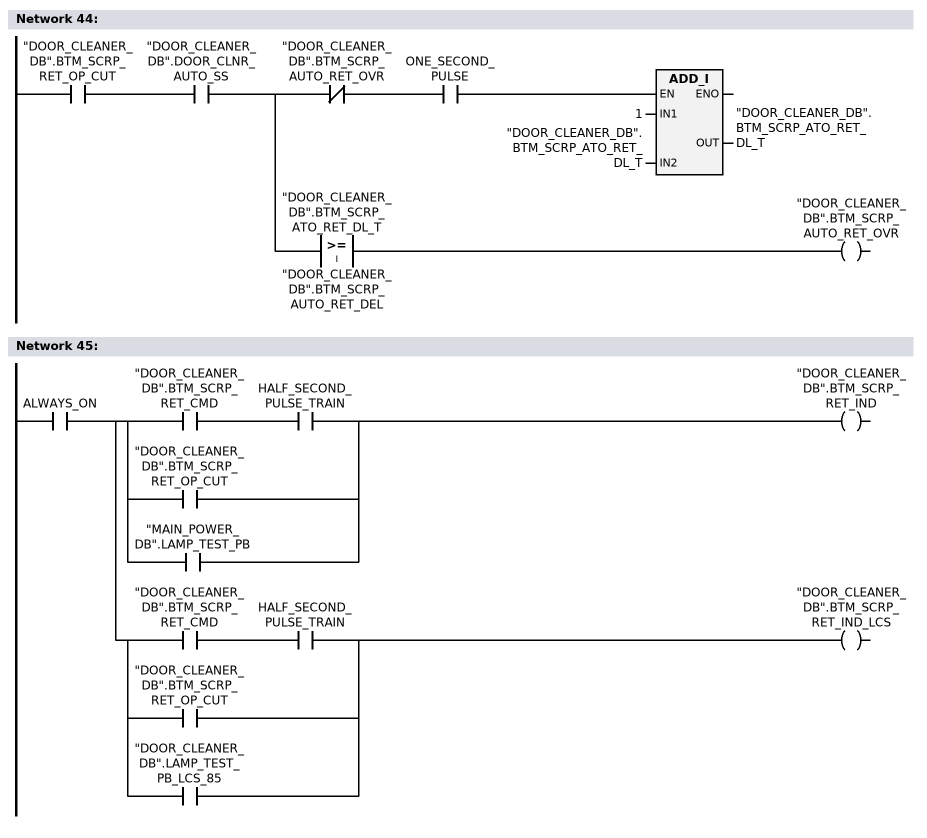
NETWORK
TITLE =
      A     "DOOR_CLEANER_DB".BTM_SCRP_RET_OP_CUT;
      A     "DOOR_CLEANER_DB".DOOR_CLNR_AUTO_SS;
      =     L 0.0;
      A     L 0.0;
      AN    "DOOR_CLEANER_DB".BTM_SCRP_AUTO_RET_OVR;
      A     "ONE_SECOND_PULSE";
      JNB   M042;
      L     1;
      L     "DOOR_CLEANER_DB".BTM_SCRP_ATO_RET_DL_T;
      +I;
      T     "DOOR_CLEANER_DB".BTM_SCRP_ATO_RET_DL_T;
M042: NOP   0;
      A     L 0.0;
      A(;
      L     "DOOR_CLEANER_DB".BTM_SCRP_ATO_RET_DL_T;
      L     "DOOR_CLEANER_DB".BTM_SCRP_AUTO_RET_DEL;
      >=I;
      );
      =     "DOOR_CLEANER_DB".BTM_SCRP_AUTO_RET_OVR;
NETWORK
TITLE =
      A     "ALWAYS_ON";
      =     L 0.0;
      A     L 0.0;
      A(;
      A     "DOOR_CLEANER_DB".BTM_SCRP_RET_CMD;
      A     "HALF_SECOND_PULSE_TRAIN";
      O     "DOOR_CLEANER_DB".BTM_SCRP_RET_OP_CUT;
      O     "MAIN_POWER_DB".LAMP_TEST_PB;
      );
      =     "DOOR_CLEANER_DB".BTM_SCRP_RET_IND;
      A     L 0.0;
      A(;
      A     "DOOR_CLEANER_DB".BTM_SCRP_RET_CMD;
      A     "HALF_SECOND_PULSE_TRAIN";
      O     "DOOR_CLEANER_DB".BTM_SCRP_RET_OP_CUT;
      O     "DOOR_CLEANER_DB".LAMP_TEST_PB_LCS_85;
      );
      =     "DOOR_CLEANER_DB".BTM_SCRP_RET_IND_LCS;
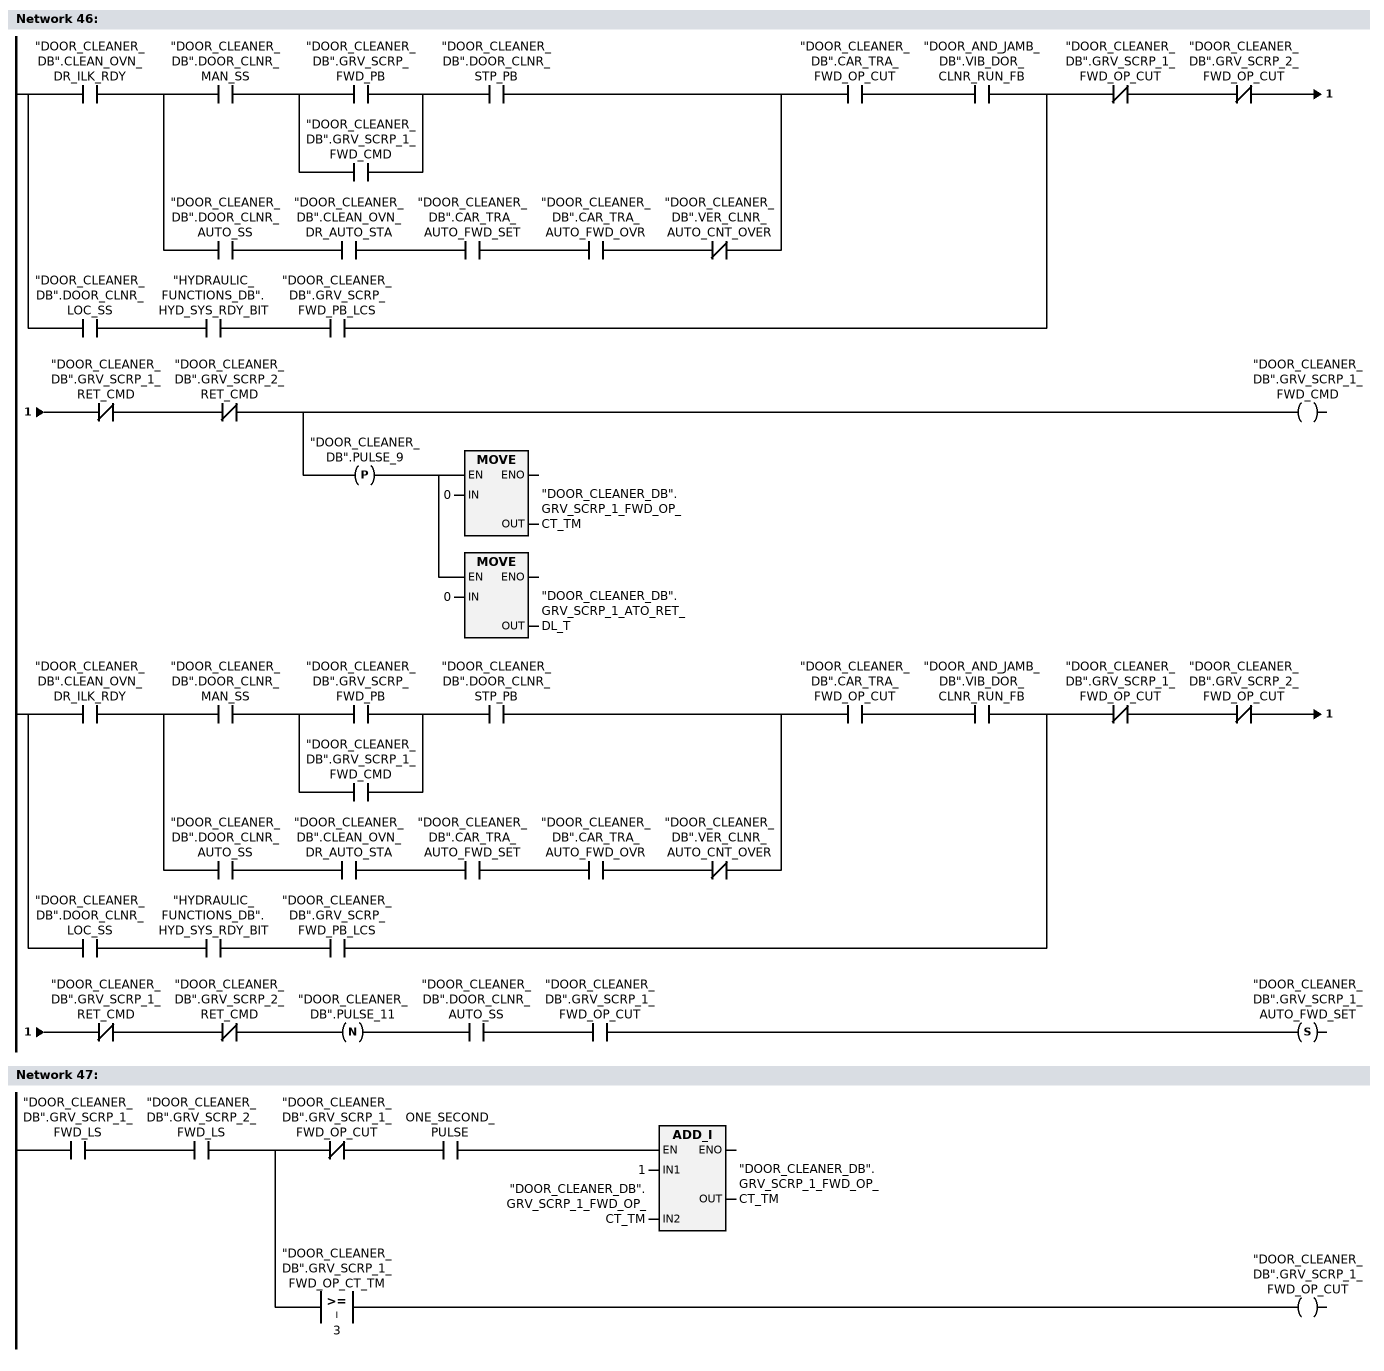
NETWORK
TITLE =
      A(;
      A     "DOOR_CLEANER_DB".CLEAN_OVN_DR_ILK_RDY;
      A(;
      A     "DOOR_CLEANER_DB".DOOR_CLNR_MAN_SS;
      A(;
      O     "DOOR_CLEANER_DB".GRV_SCRP_FWD_PB;
      O     "DOOR_CLEANER_DB".GRV_SCRP_1_FWD_CMD;
      );
      A     "DOOR_CLEANER_DB".DOOR_CLNR_STP_PB;
      O;
      A     "DOOR_CLEANER_DB".DOOR_CLNR_AUTO_SS;
      A     "DOOR_CLEANER_DB".CLEAN_OVN_DR_AUTO_STA;
      A     "DOOR_CLEANER_DB".CAR_TRA_AUTO_FWD_SET;
      A     "DOOR_CLEANER_DB".CAR_TRA_AUTO_FWD_OVR;
      AN    "DOOR_CLEANER_DB".VER_CLNR_AUTO_CNT_OVER;
      );
      A     "DOOR_CLEANER_DB".CAR_TRA_FWD_OP_CUT;
      A     "DOOR_AND_JAMB_DB".VIB_DOR_CLNR_RUN_FB;
      O;
      A     "DOOR_CLEANER_DB".DOOR_CLNR_LOC_SS;
      A     "HYDRAULIC_FUNCTIONS_DB".HYD_SYS_RDY_BIT;
      A     "DOOR_CLEANER_DB".GRV_SCRP_FWD_PB_LCS;
      );
      AN    "DOOR_CLEANER_DB".GRV_SCRP_1_FWD_OP_CUT;
      AN    "DOOR_CLEANER_DB".GRV_SCRP_2_FWD_OP_CUT;
      AN    "DOOR_CLEANER_DB".GRV_SCRP_1_RET_CMD;
      AN    "DOOR_CLEANER_DB".GRV_SCRP_2_RET_CMD;
      =     L 0.0;
      A     L 0.0;
      BLD   102;
      =     "DOOR_CLEANER_DB".GRV_SCRP_1_FWD_CMD;
      A(;
      A     L 0.0;
      FN    "DOOR_CLEANER_DB".PULSE_11;
      );
      A     "DOOR_CLEANER_DB".DOOR_CLNR_AUTO_SS;
      A     "DOOR_CLEANER_DB".GRV_SCRP_1_FWD_OP_CUT;
      S     "DOOR_CLEANER_DB".GRV_SCRP_1_AUTO_FWD_SET;
      A     L 0.0;
      FP    "DOOR_CLEANER_DB".PULSE_9;
      =     L 0.1;
      A     L 0.1;
      JNB   M043;
      L     0;
      T     "DOOR_CLEANER_DB".GRV_SCRP_1_FWD_OP_CT_TM;
M043: NOP   0;
      A     L 0.1;
      JNB   M044;
      L     0;
      T     "DOOR_CLEANER_DB".GRV_SCRP_1_ATO_RET_DL_T;
M044: NOP   0;
NETWORK
TITLE =
      A     "DOOR_CLEANER_DB".GRV_SCRP_1_FWD_LS;
      A     "DOOR_CLEANER_DB".GRV_SCRP_2_FWD_LS;
      =     L 0.0;
      A     L 0.0;
      AN    "DOOR_CLEANER_DB".GRV_SCRP_1_FWD_OP_CUT;
      A     "ONE_SECOND_PULSE";
      JNB   M045;
      L     1;
      L     "DOOR_CLEANER_DB".GRV_SCRP_1_FWD_OP_CT_TM;
      +I;
      T     "DOOR_CLEANER_DB".GRV_SCRP_1_FWD_OP_CT_TM;
M045: NOP   0;
      A     L 0.0;
      A(;
      L     "DOOR_CLEANER_DB".GRV_SCRP_1_FWD_OP_CT_TM;
      L     3;
      >=I;
      );
      =     "DOOR_CLEANER_DB".GRV_SCRP_1_FWD_OP_CUT;
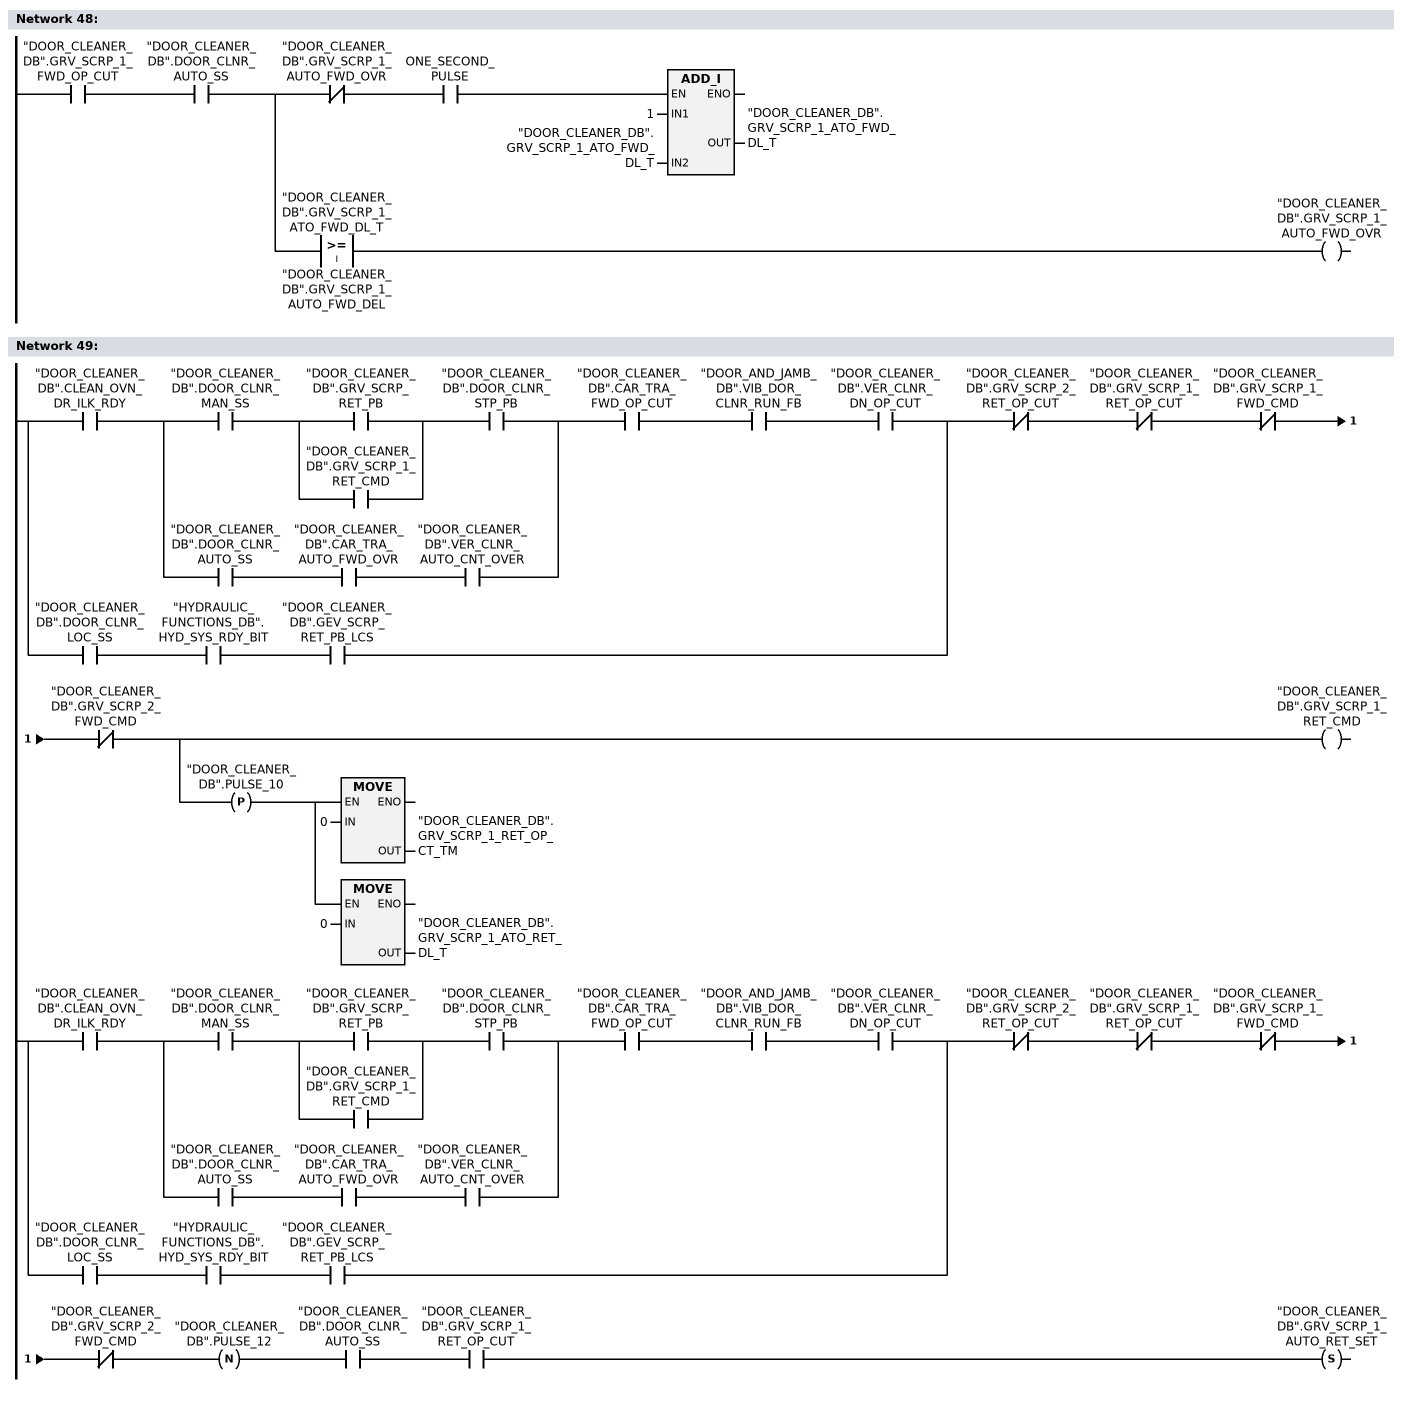
NETWORK
TITLE =
      A     "DOOR_CLEANER_DB".GRV_SCRP_1_FWD_OP_CUT;
      A     "DOOR_CLEANER_DB".DOOR_CLNR_AUTO_SS;
      =     L 0.0;
      A     L 0.0;
      AN    "DOOR_CLEANER_DB".GRV_SCRP_1_AUTO_FWD_OVR;
      A     "ONE_SECOND_PULSE";
      JNB   M046;
      L     1;
      L     "DOOR_CLEANER_DB".GRV_SCRP_1_ATO_FWD_DL_T;
      +I;
      T     "DOOR_CLEANER_DB".GRV_SCRP_1_ATO_FWD_DL_T;
M046: NOP   0;
      A     L 0.0;
      A(;
      L     "DOOR_CLEANER_DB".GRV_SCRP_1_ATO_FWD_DL_T;
      L     "DOOR_CLEANER_DB".GRV_SCRP_1_AUTO_FWD_DEL;
      >=I;
      );
      =     "DOOR_CLEANER_DB".GRV_SCRP_1_AUTO_FWD_OVR;
NETWORK
TITLE =
      A(;
      A     "DOOR_CLEANER_DB".CLEAN_OVN_DR_ILK_RDY;
      A(;
      A     "DOOR_CLEANER_DB".DOOR_CLNR_MAN_SS;
      A(;
      O     "DOOR_CLEANER_DB".GRV_SCRP_RET_PB;
      O     "DOOR_CLEANER_DB".GRV_SCRP_1_RET_CMD;
      );
      A     "DOOR_CLEANER_DB".DOOR_CLNR_STP_PB;
      O;
      A     "DOOR_CLEANER_DB".DOOR_CLNR_AUTO_SS;
      A     "DOOR_CLEANER_DB".CAR_TRA_AUTO_FWD_OVR;
      A     "DOOR_CLEANER_DB".VER_CLNR_AUTO_CNT_OVER;
      );
      A     "DOOR_CLEANER_DB".CAR_TRA_FWD_OP_CUT;
      A     "DOOR_AND_JAMB_DB".VIB_DOR_CLNR_RUN_FB;
      A     "DOOR_CLEANER_DB".VER_CLNR_DN_OP_CUT;
      O;
      A     "DOOR_CLEANER_DB".DOOR_CLNR_LOC_SS;
      A     "HYDRAULIC_FUNCTIONS_DB".HYD_SYS_RDY_BIT;
      A     "DOOR_CLEANER_DB".GEV_SCRP_RET_PB_LCS;
      );
      AN    "DOOR_CLEANER_DB".GRV_SCRP_2_RET_OP_CUT;
      AN    "DOOR_CLEANER_DB".GRV_SCRP_1_RET_OP_CUT;
      AN    "DOOR_CLEANER_DB".GRV_SCRP_1_FWD_CMD;
      AN    "DOOR_CLEANER_DB".GRV_SCRP_2_FWD_CMD;
      =     L 0.0;
      A     L 0.0;
      BLD   102;
      =     "DOOR_CLEANER_DB".GRV_SCRP_1_RET_CMD;
      A(;
      A     L 0.0;
      FN    "DOOR_CLEANER_DB".PULSE_12;
      );
      A     "DOOR_CLEANER_DB".DOOR_CLNR_AUTO_SS;
      A     "DOOR_CLEANER_DB".GRV_SCRP_1_RET_OP_CUT;
      S     "DOOR_CLEANER_DB".GRV_SCRP_1_AUTO_RET_SET;
      A     L 0.0;
      FP    "DOOR_CLEANER_DB".PULSE_10;
      =     L 0.1;
      A     L 0.1;
      JNB   M047;
      L     0;
      T     "DOOR_CLEANER_DB".GRV_SCRP_1_RET_OP_CT_TM;
M047: NOP   0;
      A     L 0.1;
      JNB   M048;
      L     0;
      T     "DOOR_CLEANER_DB".GRV_SCRP_1_ATO_RET_DL_T;
M048: NOP   0;
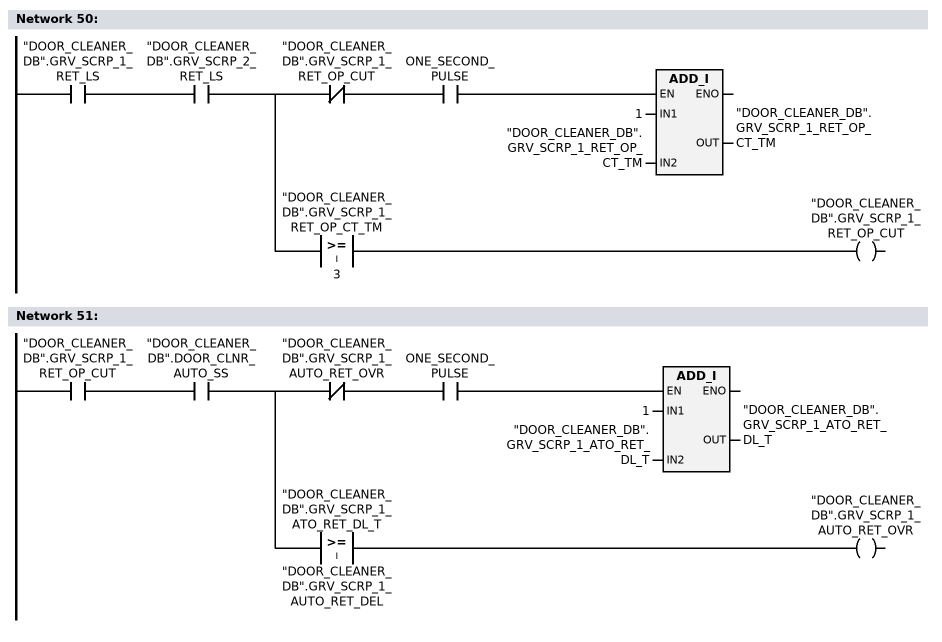
NETWORK
TITLE =
      A     "DOOR_CLEANER_DB".GRV_SCRP_1_RET_LS;
      A     "DOOR_CLEANER_DB".GRV_SCRP_2_RET_LS;
      =     L 0.0;
      A     L 0.0;
      AN    "DOOR_CLEANER_DB".GRV_SCRP_1_RET_OP_CUT;
      A     "ONE_SECOND_PULSE";
      JNB   M049;
      L     1;
      L     "DOOR_CLEANER_DB".GRV_SCRP_1_RET_OP_CT_TM;
      +I;
      T     "DOOR_CLEANER_DB".GRV_SCRP_1_RET_OP_CT_TM;
M049: NOP   0;
      A     L 0.0;
      A(;
      L     "DOOR_CLEANER_DB".GRV_SCRP_1_RET_OP_CT_TM;
      L     3;
      >=I;
      );
      =     "DOOR_CLEANER_DB".GRV_SCRP_1_RET_OP_CUT;
NETWORK
TITLE =
      A     "DOOR_CLEANER_DB".GRV_SCRP_1_RET_OP_CUT;
      A     "DOOR_CLEANER_DB".DOOR_CLNR_AUTO_SS;
      =     L 0.0;
      A     L 0.0;
      AN    "DOOR_CLEANER_DB".GRV_SCRP_1_AUTO_RET_OVR;
      A     "ONE_SECOND_PULSE";
      JNB   M050;
      L     1;
      L     "DOOR_CLEANER_DB".GRV_SCRP_1_ATO_RET_DL_T;
      +I;
      T     "DOOR_CLEANER_DB".GRV_SCRP_1_ATO_RET_DL_T;
M050: NOP   0;
      A     L 0.0;
      A(;
      L     "DOOR_CLEANER_DB".GRV_SCRP_1_ATO_RET_DL_T;
      L     "DOOR_CLEANER_DB".GRV_SCRP_1_AUTO_RET_DEL;
      >=I;
      );
      =     "DOOR_CLEANER_DB".GRV_SCRP_1_AUTO_RET_OVR;
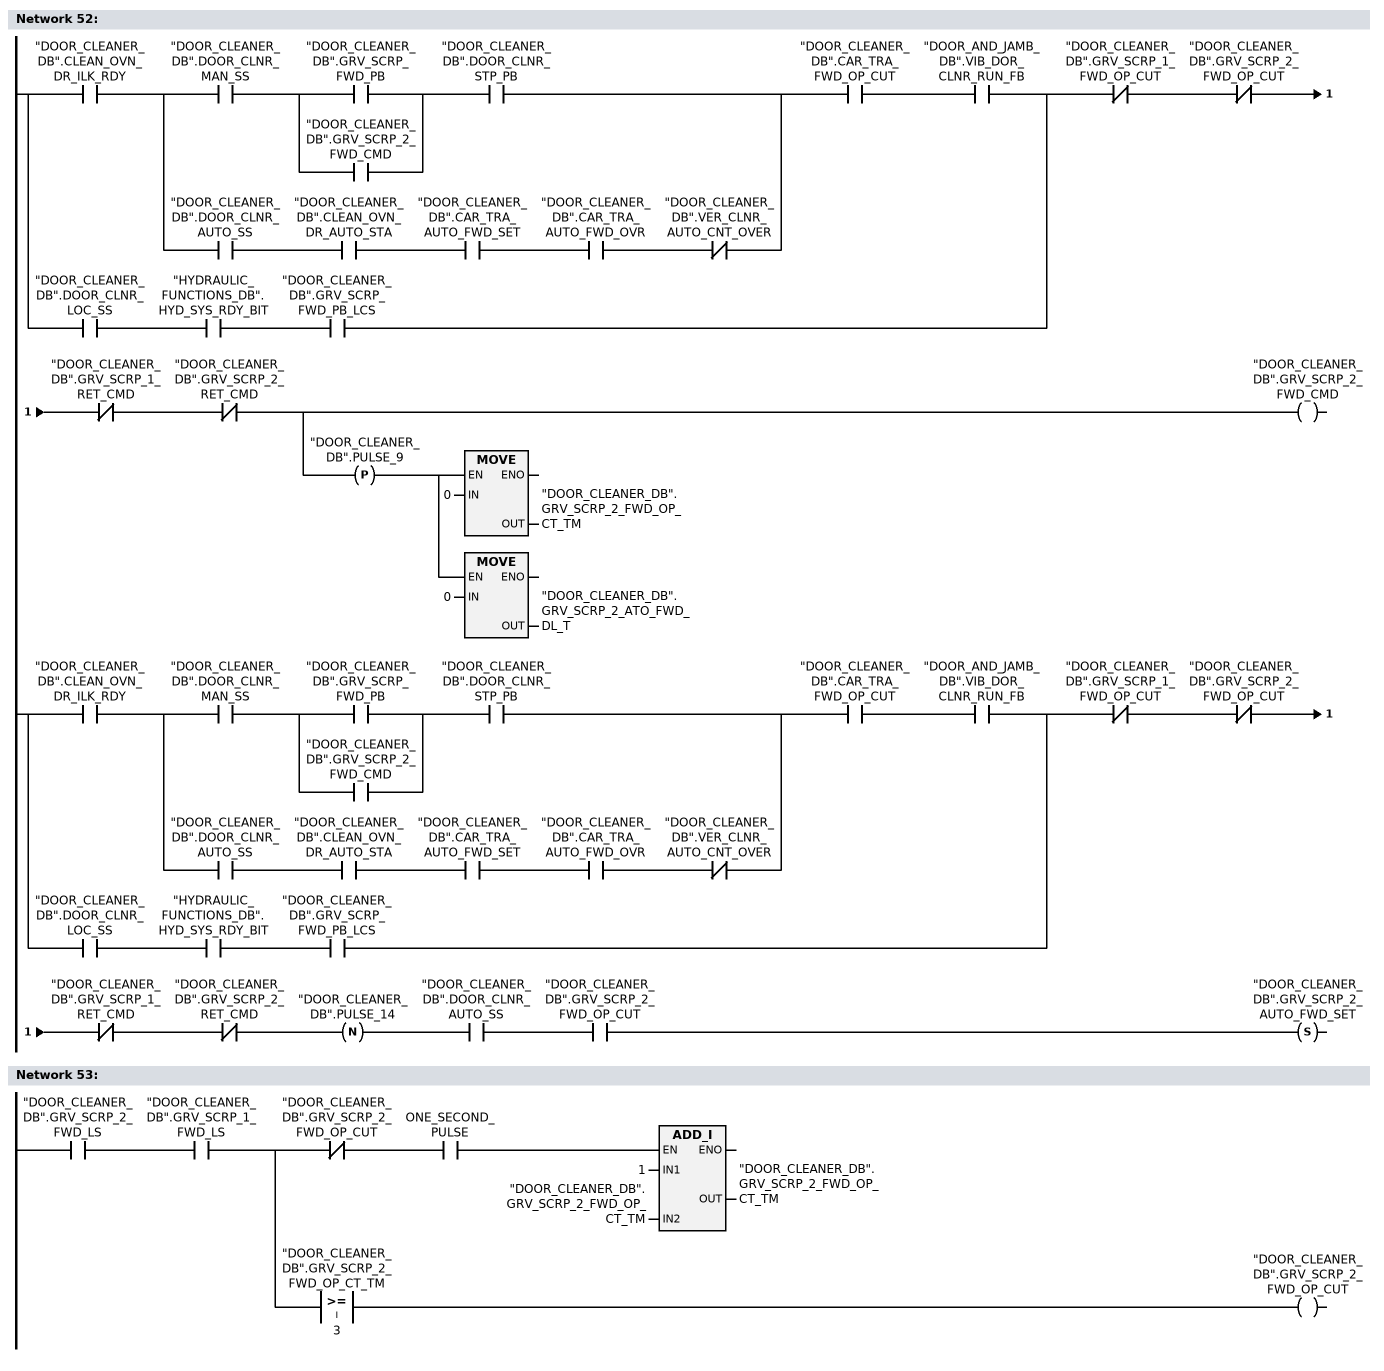
NETWORK
TITLE =
      A(;
      A     "DOOR_CLEANER_DB".CLEAN_OVN_DR_ILK_RDY;
      A(;
      A     "DOOR_CLEANER_DB".DOOR_CLNR_MAN_SS;
      A(;
      O     "DOOR_CLEANER_DB".GRV_SCRP_FWD_PB;
      O     "DOOR_CLEANER_DB".GRV_SCRP_2_FWD_CMD;
      );
      A     "DOOR_CLEANER_DB".DOOR_CLNR_STP_PB;
      O;
      A     "DOOR_CLEANER_DB".DOOR_CLNR_AUTO_SS;
      A     "DOOR_CLEANER_DB".CLEAN_OVN_DR_AUTO_STA;
      A     "DOOR_CLEANER_DB".CAR_TRA_AUTO_FWD_SET;
      A     "DOOR_CLEANER_DB".CAR_TRA_AUTO_FWD_OVR;
      AN    "DOOR_CLEANER_DB".VER_CLNR_AUTO_CNT_OVER;
      );
      A     "DOOR_CLEANER_DB".CAR_TRA_FWD_OP_CUT;
      A     "DOOR_AND_JAMB_DB".VIB_DOR_CLNR_RUN_FB;
      O;
      A     "DOOR_CLEANER_DB".DOOR_CLNR_LOC_SS;
      A     "HYDRAULIC_FUNCTIONS_DB".HYD_SYS_RDY_BIT;
      A     "DOOR_CLEANER_DB".GRV_SCRP_FWD_PB_LCS;
      );
      AN    "DOOR_CLEANER_DB".GRV_SCRP_1_FWD_OP_CUT;
      AN    "DOOR_CLEANER_DB".GRV_SCRP_2_FWD_OP_CUT;
      AN    "DOOR_CLEANER_DB".GRV_SCRP_1_RET_CMD;
      AN    "DOOR_CLEANER_DB".GRV_SCRP_2_RET_CMD;
      =     L 0.0;
      A     L 0.0;
      BLD   102;
      =     "DOOR_CLEANER_DB".GRV_SCRP_2_FWD_CMD;
      A(;
      A     L 0.0;
      FN    "DOOR_CLEANER_DB".PULSE_14;
      );
      A     "DOOR_CLEANER_DB".DOOR_CLNR_AUTO_SS;
      A     "DOOR_CLEANER_DB".GRV_SCRP_2_FWD_OP_CUT;
      S     "DOOR_CLEANER_DB".GRV_SCRP_2_AUTO_FWD_SET;
      A     L 0.0;
      FP    "DOOR_CLEANER_DB".PULSE_9;
      =     L 0.1;
      A     L 0.1;
      JNB   M051;
      L     0;
      T     "DOOR_CLEANER_DB".GRV_SCRP_2_FWD_OP_CT_TM;
M051: NOP   0;
      A     L 0.1;
      JNB   M052;
      L     0;
      T     "DOOR_CLEANER_DB".GRV_SCRP_2_ATO_FWD_DL_T;
M052: NOP   0;
NETWORK
TITLE =
      A     "DOOR_CLEANER_DB".GRV_SCRP_2_FWD_LS;
      A     "DOOR_CLEANER_DB".GRV_SCRP_1_FWD_LS;
      =     L 0.0;
      A     L 0.0;
      AN    "DOOR_CLEANER_DB".GRV_SCRP_2_FWD_OP_CUT;
      A     "ONE_SECOND_PULSE";
      JNB   M053;
      L     1;
      L     "DOOR_CLEANER_DB".GRV_SCRP_2_FWD_OP_CT_TM;
      +I;
      T     "DOOR_CLEANER_DB".GRV_SCRP_2_FWD_OP_CT_TM;
M053: NOP   0;
      A     L 0.0;
      A(;
      L     "DOOR_CLEANER_DB".GRV_SCRP_2_FWD_OP_CT_TM;
      L     3;
      >=I;
      );
      =     "DOOR_CLEANER_DB".GRV_SCRP_2_FWD_OP_CUT;
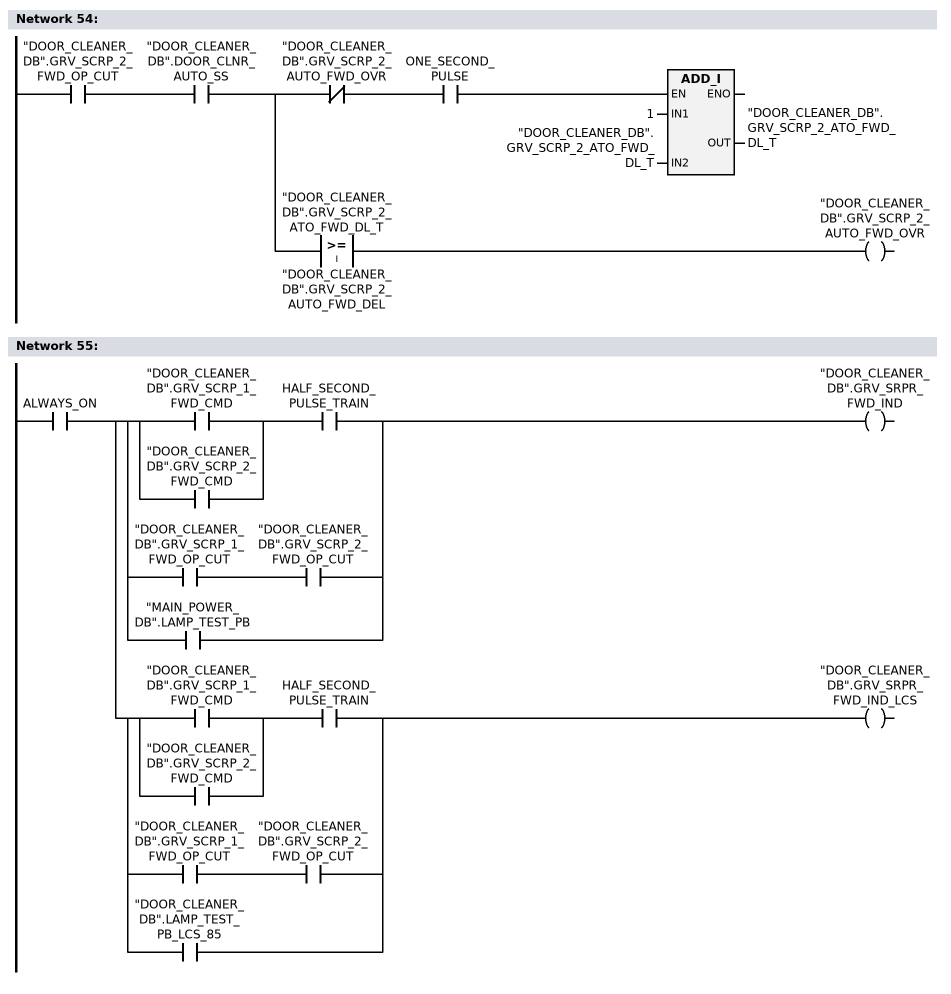
NETWORK
TITLE =
      A     "DOOR_CLEANER_DB".GRV_SCRP_2_FWD_OP_CUT;
      A     "DOOR_CLEANER_DB".DOOR_CLNR_AUTO_SS;
      =     L 0.0;
      A     L 0.0;
      AN    "DOOR_CLEANER_DB".GRV_SCRP_2_AUTO_FWD_OVR;
      A     "ONE_SECOND_PULSE";
      JNB   M054;
      L     1;
      L     "DOOR_CLEANER_DB".GRV_SCRP_2_ATO_FWD_DL_T;
      +I;
      T     "DOOR_CLEANER_DB".GRV_SCRP_2_ATO_FWD_DL_T;
M054: NOP   0;
      A     L 0.0;
      A(;
      L     "DOOR_CLEANER_DB".GRV_SCRP_2_ATO_FWD_DL_T;
      L     "DOOR_CLEANER_DB".GRV_SCRP_2_AUTO_FWD_DEL;
      >=I;
      );
      =     "DOOR_CLEANER_DB".GRV_SCRP_2_AUTO_FWD_OVR;
NETWORK
TITLE =
      A     "ALWAYS_ON";
      =     L 0.0;
      A     L 0.0;
      A(;
      A(;
      O     "DOOR_CLEANER_DB".GRV_SCRP_1_FWD_CMD;
      O     "DOOR_CLEANER_DB".GRV_SCRP_2_FWD_CMD;
      );
      A     "HALF_SECOND_PULSE_TRAIN";
      O;
      A     "DOOR_CLEANER_DB".GRV_SCRP_1_FWD_OP_CUT;
      A     "DOOR_CLEANER_DB".GRV_SCRP_2_FWD_OP_CUT;
      O     "MAIN_POWER_DB".LAMP_TEST_PB;
      );
      =     "DOOR_CLEANER_DB".GRV_SRPR_FWD_IND;
      A     L 0.0;
      A(;
      A(;
      O     "DOOR_CLEANER_DB".GRV_SCRP_1_FWD_CMD;
      O     "DOOR_CLEANER_DB".GRV_SCRP_2_FWD_CMD;
      );
      A     "HALF_SECOND_PULSE_TRAIN";
      O;
      A     "DOOR_CLEANER_DB".GRV_SCRP_1_FWD_OP_CUT;
      A     "DOOR_CLEANER_DB".GRV_SCRP_2_FWD_OP_CUT;
      O     "DOOR_CLEANER_DB".LAMP_TEST_PB_LCS_85;
      );
      =     "DOOR_CLEANER_DB".GRV_SRPR_FWD_IND_LCS;
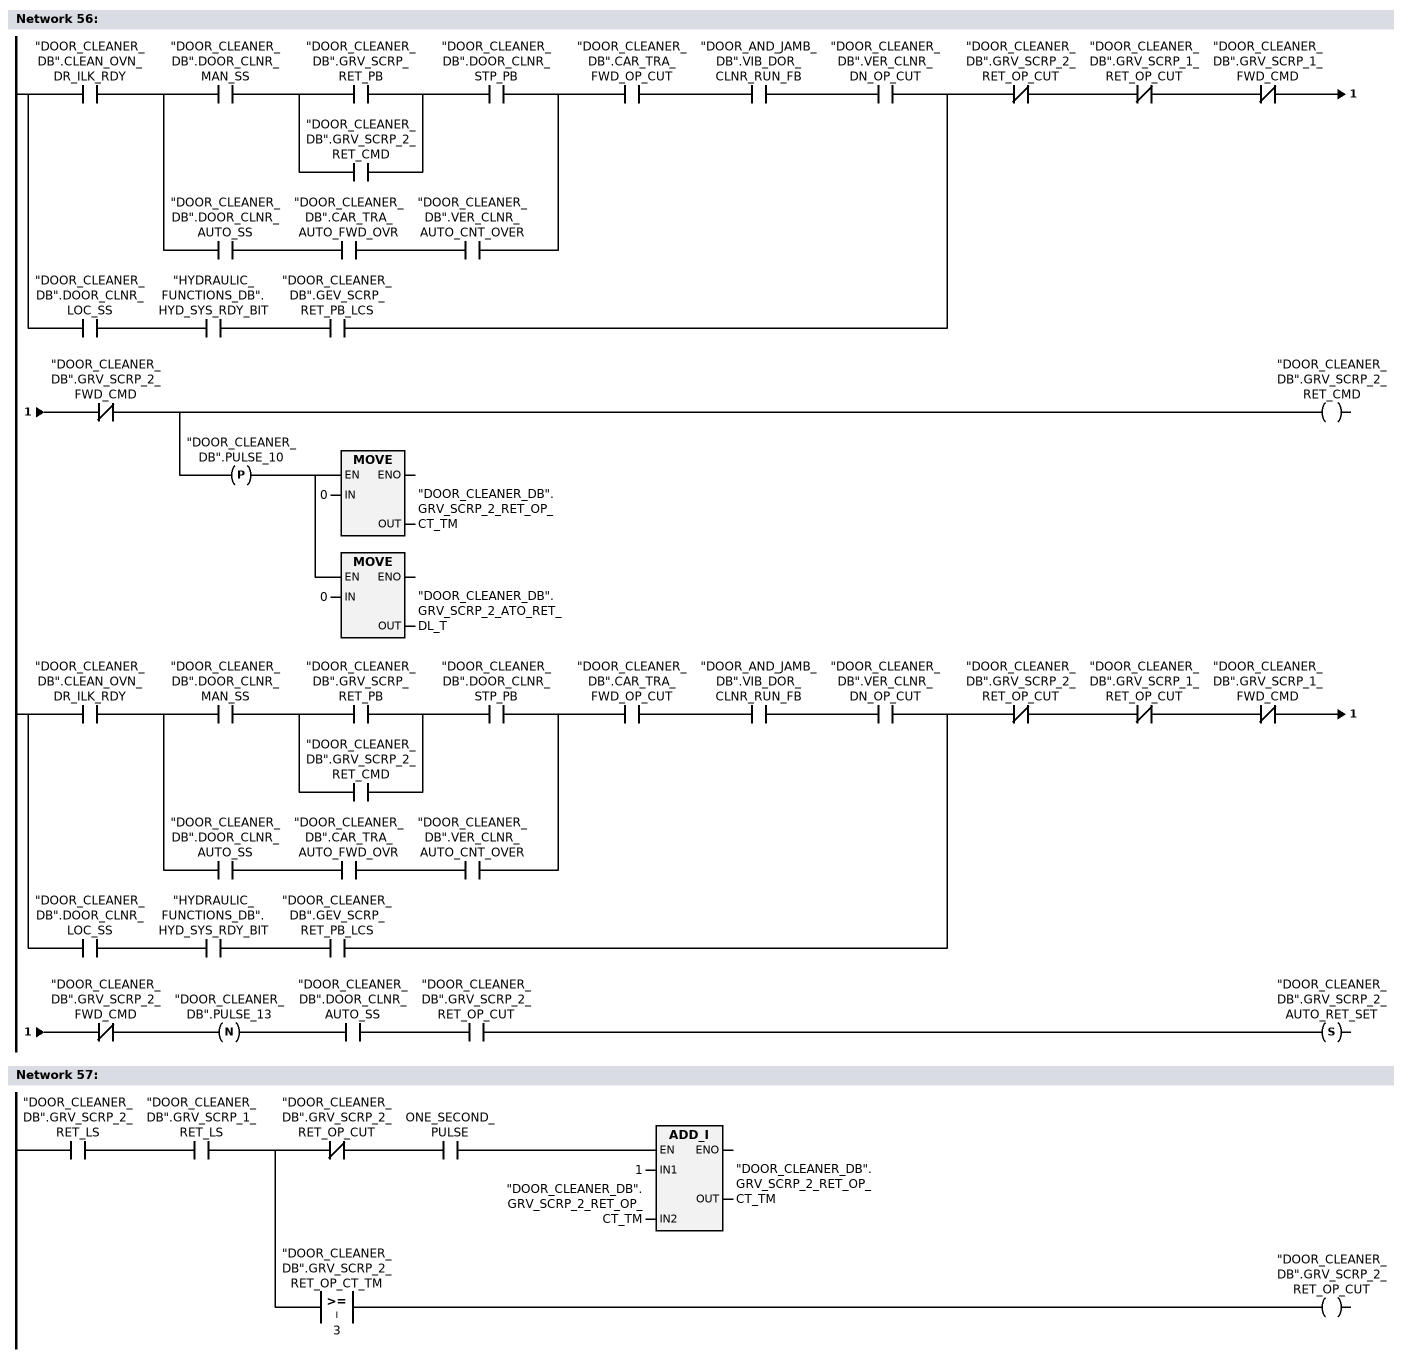
NETWORK
TITLE =
      A(;
      A     "DOOR_CLEANER_DB".CLEAN_OVN_DR_ILK_RDY;
      A(;
      A     "DOOR_CLEANER_DB".DOOR_CLNR_MAN_SS;
      A(;
      O     "DOOR_CLEANER_DB".GRV_SCRP_RET_PB;
      O     "DOOR_CLEANER_DB".GRV_SCRP_2_RET_CMD;
      );
      A     "DOOR_CLEANER_DB".DOOR_CLNR_STP_PB;
      O;
      A     "DOOR_CLEANER_DB".DOOR_CLNR_AUTO_SS;
      A     "DOOR_CLEANER_DB".CAR_TRA_AUTO_FWD_OVR;
      A     "DOOR_CLEANER_DB".VER_CLNR_AUTO_CNT_OVER;
      );
      A     "DOOR_CLEANER_DB".CAR_TRA_FWD_OP_CUT;
      A     "DOOR_AND_JAMB_DB".VIB_DOR_CLNR_RUN_FB;
      A     "DOOR_CLEANER_DB".VER_CLNR_DN_OP_CUT;
      O;
      A     "DOOR_CLEANER_DB".DOOR_CLNR_LOC_SS;
      A     "HYDRAULIC_FUNCTIONS_DB".HYD_SYS_RDY_BIT;
      A     "DOOR_CLEANER_DB".GEV_SCRP_RET_PB_LCS;
      );
      AN    "DOOR_CLEANER_DB".GRV_SCRP_2_RET_OP_CUT;
      AN    "DOOR_CLEANER_DB".GRV_SCRP_1_RET_OP_CUT;
      AN    "DOOR_CLEANER_DB".GRV_SCRP_1_FWD_CMD;
      AN    "DOOR_CLEANER_DB".GRV_SCRP_2_FWD_CMD;
      =     L 0.0;
      A     L 0.0;
      BLD   102;
      =     "DOOR_CLEANER_DB".GRV_SCRP_2_RET_CMD;
      A(;
      A     L 0.0;
      FN    "DOOR_CLEANER_DB".PULSE_13;
      );
      A     "DOOR_CLEANER_DB".DOOR_CLNR_AUTO_SS;
      A     "DOOR_CLEANER_DB".GRV_SCRP_2_RET_OP_CUT;
      S     "DOOR_CLEANER_DB".GRV_SCRP_2_AUTO_RET_SET;
      A     L 0.0;
      FP    "DOOR_CLEANER_DB".PULSE_10;
      =     L 0.1;
      A     L 0.1;
      JNB   M055;
      L     0;
      T     "DOOR_CLEANER_DB".GRV_SCRP_2_RET_OP_CT_TM;
M055: NOP   0;
      A     L 0.1;
      JNB   M056;
      L     0;
      T     "DOOR_CLEANER_DB".GRV_SCRP_2_ATO_RET_DL_T;
M056: NOP   0;
NETWORK
TITLE =
      A     "DOOR_CLEANER_DB".GRV_SCRP_2_RET_LS;
      A     "DOOR_CLEANER_DB".GRV_SCRP_1_RET_LS;
      =     L 0.0;
      A     L 0.0;
      AN    "DOOR_CLEANER_DB".GRV_SCRP_2_RET_OP_CUT;
      A     "ONE_SECOND_PULSE";
      JNB   M057;
      L     1;
      L     "DOOR_CLEANER_DB".GRV_SCRP_2_RET_OP_CT_TM;
      +I;
      T     "DOOR_CLEANER_DB".GRV_SCRP_2_RET_OP_CT_TM;
M057: NOP   0;
      A     L 0.0;
      A(;
      L     "DOOR_CLEANER_DB".GRV_SCRP_2_RET_OP_CT_TM;
      L     3;
      >=I;
      );
      =     "DOOR_CLEANER_DB".GRV_SCRP_2_RET_OP_CUT;
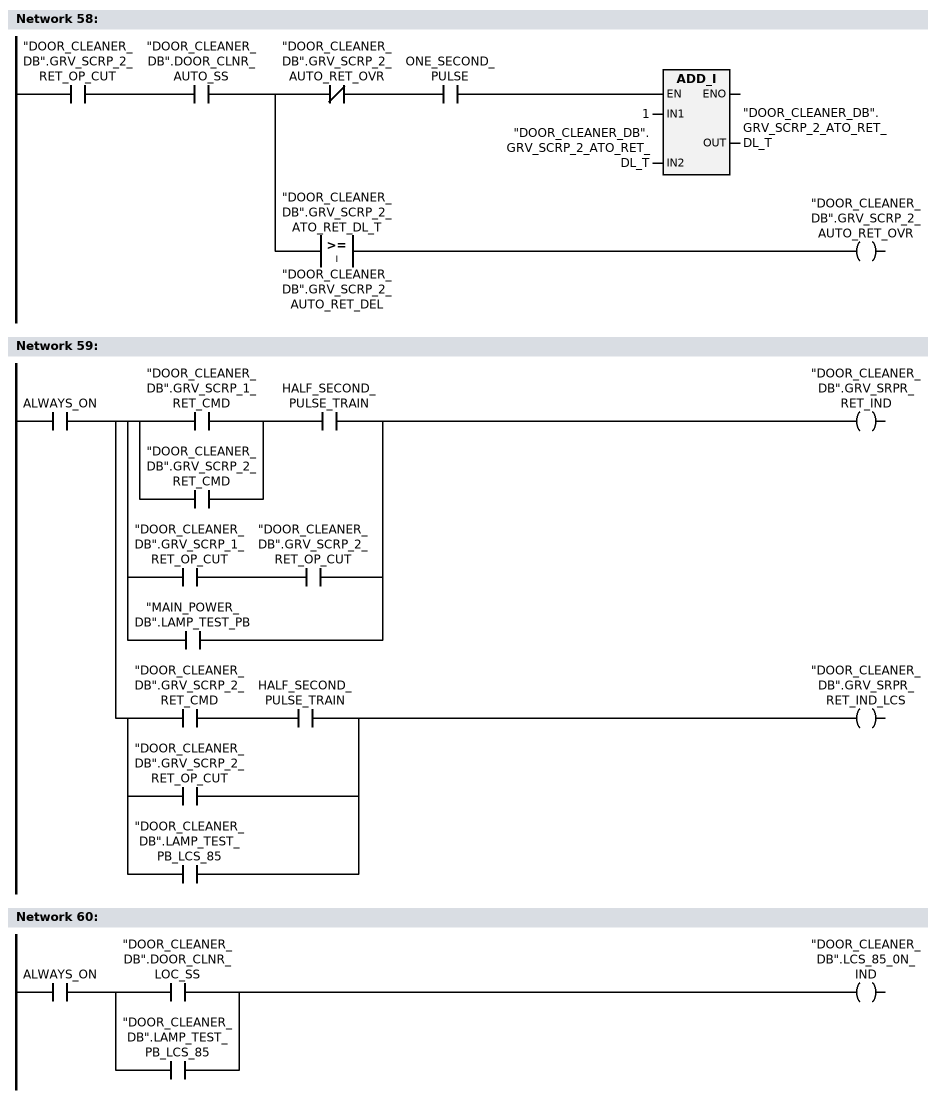
NETWORK
TITLE =
      A     "DOOR_CLEANER_DB".GRV_SCRP_2_RET_OP_CUT;
      A     "DOOR_CLEANER_DB".DOOR_CLNR_AUTO_SS;
      =     L 0.0;
      A     L 0.0;
      AN    "DOOR_CLEANER_DB".GRV_SCRP_2_AUTO_RET_OVR;
      A     "ONE_SECOND_PULSE";
      JNB   M058;
      L     1;
      L     "DOOR_CLEANER_DB".GRV_SCRP_2_ATO_RET_DL_T;
      +I;
      T     "DOOR_CLEANER_DB".GRV_SCRP_2_ATO_RET_DL_T;
M058: NOP   0;
      A     L 0.0;
      A(;
      L     "DOOR_CLEANER_DB".GRV_SCRP_2_ATO_RET_DL_T;
      L     "DOOR_CLEANER_DB".GRV_SCRP_2_AUTO_RET_DEL;
      >=I;
      );
      =     "DOOR_CLEANER_DB".GRV_SCRP_2_AUTO_RET_OVR;
NETWORK
TITLE =
      A     "ALWAYS_ON";
      =     L 0.0;
      A     L 0.0;
      A(;
      A(;
      O     "DOOR_CLEANER_DB".GRV_SCRP_1_RET_CMD;
      O     "DOOR_CLEANER_DB".GRV_SCRP_2_RET_CMD;
      );
      A     "HALF_SECOND_PULSE_TRAIN";
      O;
      A     "DOOR_CLEANER_DB".GRV_SCRP_1_RET_OP_CUT;
      A     "DOOR_CLEANER_DB".GRV_SCRP_2_RET_OP_CUT;
      O     "MAIN_POWER_DB".LAMP_TEST_PB;
      );
      =     "DOOR_CLEANER_DB".GRV_SRPR_RET_IND;
      A     L 0.0;
      A(;
      A     "DOOR_CLEANER_DB".GRV_SCRP_2_RET_CMD;
      A     "HALF_SECOND_PULSE_TRAIN";
      O     "DOOR_CLEANER_DB".GRV_SCRP_2_RET_OP_CUT;
      O     "DOOR_CLEANER_DB".LAMP_TEST_PB_LCS_85;
      );
      =     "DOOR_CLEANER_DB".GRV_SRPR_RET_IND_LCS;
NETWORK
TITLE =
      A     "ALWAYS_ON";
      A(;
      O     "DOOR_CLEANER_DB".DOOR_CLNR_LOC_SS;
      O     "DOOR_CLEANER_DB".LAMP_TEST_PB_LCS_85;
      );
      =     "DOOR_CLEANER_DB".LCS_85_0N_IND;
END_FUNCTION

FUNCTION "JAMB_CLEANER" : VOID	// FC 16
AUTHOR : Kamillas
VERSION : 0.1
BEGIN
// (block stored without names or comments; labels and parameter names are numbered)
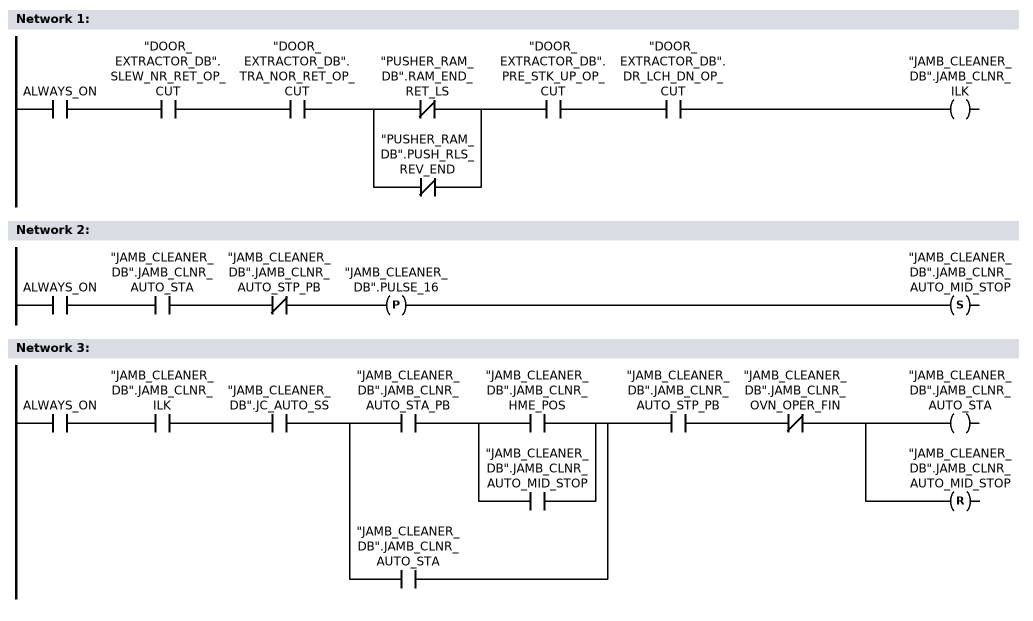
NETWORK
TITLE =
      A     "ALWAYS_ON";
      A     "DOOR_EXTRACTOR_DB".SLEW_NR_RET_OP_CUT;
      A     "DOOR_EXTRACTOR_DB".TRA_NOR_RET_OP_CUT;
      A(;
      ON    "PUSHER_RAM_DB".RAM_END_RET_LS;
      ON    "PUSHER_RAM_DB".PUSH_RLS_REV_END;
      );
      A     "DOOR_EXTRACTOR_DB".PRE_STK_UP_OP_CUT;
      A     "DOOR_EXTRACTOR_DB".DR_LCH_DN_OP_CUT;
      =     "JAMB_CLEANER_DB".JAMB_CLNR_ILK;
NETWORK
TITLE =
      A     "ALWAYS_ON";
      A     "JAMB_CLEANER_DB".JAMB_CLNR_AUTO_STA;
      AN    "JAMB_CLEANER_DB".JAMB_CLNR_AUTO_STP_PB;
      FP    "JAMB_CLEANER_DB".PULSE_16;
      S     "JAMB_CLEANER_DB".JAMB_CLNR_AUTO_MID_STOP;
NETWORK
TITLE =
      A     "ALWAYS_ON";
      A     "JAMB_CLEANER_DB".JAMB_CLNR_ILK;
      A     "JAMB_CLEANER_DB".JC_AUTO_SS;
      A(;
      A     "JAMB_CLEANER_DB".JAMB_CLNR_AUTO_STA_PB;
      A(;
      O     "JAMB_CLEANER_DB".JAMB_CLNR_HME_POS;
      O     "JAMB_CLEANER_DB".JAMB_CLNR_AUTO_MID_STOP;
      );
      O     "JAMB_CLEANER_DB".JAMB_CLNR_AUTO_STA;
      );
      A     "JAMB_CLEANER_DB".JAMB_CLNR_AUTO_STP_PB;
      AN    "JAMB_CLEANER_DB".JAMB_CLNR_OVN_OPER_FIN;
      =     "JAMB_CLEANER_DB".JAMB_CLNR_AUTO_STA;
      R     "JAMB_CLEANER_DB".JAMB_CLNR_AUTO_MID_STOP;
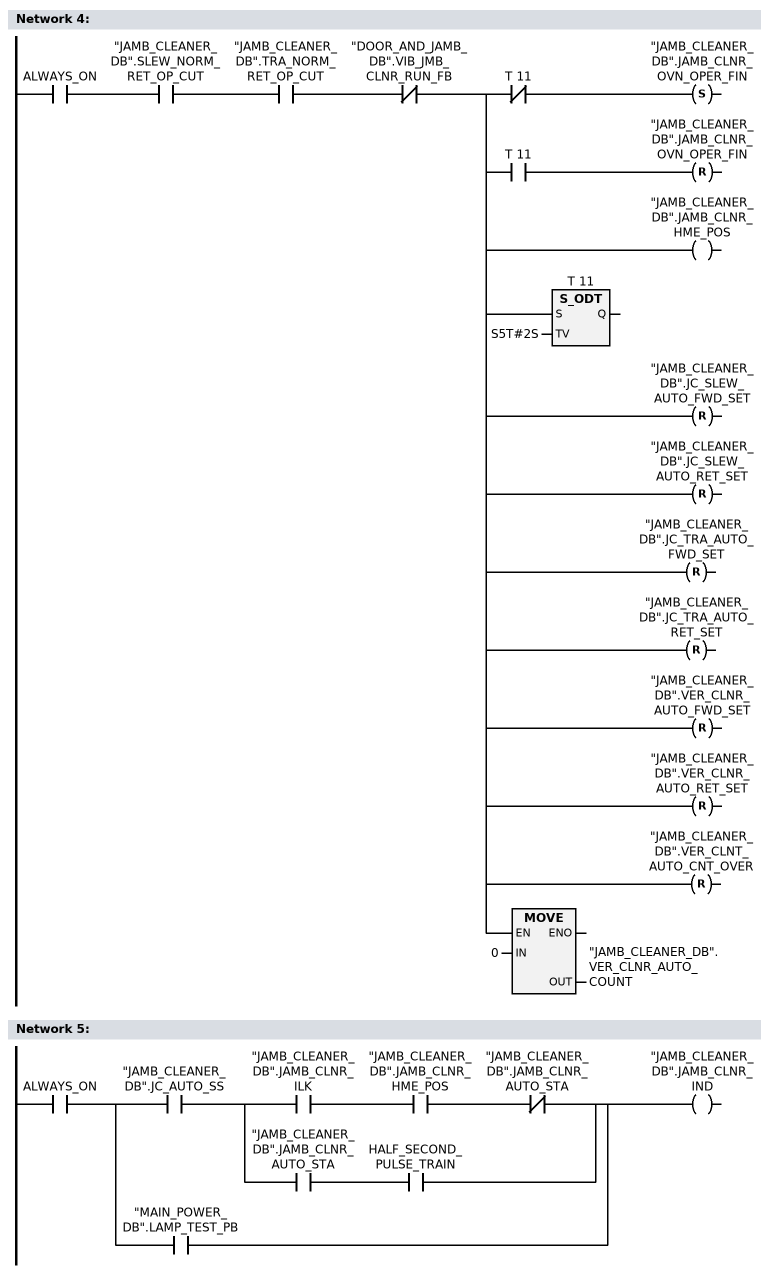
NETWORK
TITLE =
      A     "ALWAYS_ON";
      A     "JAMB_CLEANER_DB".SLEW_NORM_RET_OP_CUT;
      A     "JAMB_CLEANER_DB".TRA_NORM_RET_OP_CUT;
      AN    "DOOR_AND_JAMB_DB".VIB_JMB_CLNR_RUN_FB;
      =     L 0.0;
      A     L 0.0;
      AN    T 11;
      S     "JAMB_CLEANER_DB".JAMB_CLNR_OVN_OPER_FIN;
      A     L 0.0;
      A     T 11;
      R     "JAMB_CLEANER_DB".JAMB_CLNR_OVN_OPER_FIN;
      A     L 0.0;
      BLD   102;
      =     "JAMB_CLEANER_DB".JAMB_CLNR_HME_POS;
      A     L 0.0;
      L     S5T#2S;
      SD    T 11;
      NOP   0;
      NOP   0;
      NOP   0;
      NOP   0;
      A     L 0.0;
      BLD   102;
      R     "JAMB_CLEANER_DB".JC_SLEW_AUTO_FWD_SET;
      A     L 0.0;
      BLD   102;
      R     "JAMB_CLEANER_DB".JC_SLEW_AUTO_RET_SET;
      A     L 0.0;
      BLD   102;
      R     "JAMB_CLEANER_DB".JC_TRA_AUTO_FWD_SET;
      A     L 0.0;
      BLD   102;
      R     "JAMB_CLEANER_DB".JC_TRA_AUTO_RET_SET;
      A     L 0.0;
      BLD   102;
      R     "JAMB_CLEANER_DB".VER_CLNR_AUTO_FWD_SET;
      A     L 0.0;
      BLD   102;
      R     "JAMB_CLEANER_DB".VER_CLNR_AUTO_RET_SET;
      A     L 0.0;
      BLD   102;
      R     "JAMB_CLEANER_DB".VER_CLNT_AUTO_CNT_OVER;
      A     L 0.0;
      JNB   M001;
      L     0;
      T     "JAMB_CLEANER_DB".VER_CLNR_AUTO_COUNT;
M001: NOP   0;
NETWORK
TITLE =
      A     "ALWAYS_ON";
      A(;
      A     "JAMB_CLEANER_DB".JC_AUTO_SS;
      A(;
      A     "JAMB_CLEANER_DB".JAMB_CLNR_ILK;
      A     "JAMB_CLEANER_DB".JAMB_CLNR_HME_POS;
      AN    "JAMB_CLEANER_DB".JAMB_CLNR_AUTO_STA;
      O;
      A     "JAMB_CLEANER_DB".JAMB_CLNR_AUTO_STA;
      A     "HALF_SECOND_PULSE_TRAIN";
      );
      O     "MAIN_POWER_DB".LAMP_TEST_PB;
      );
      =     "JAMB_CLEANER_DB".JAMB_CLNR_IND;
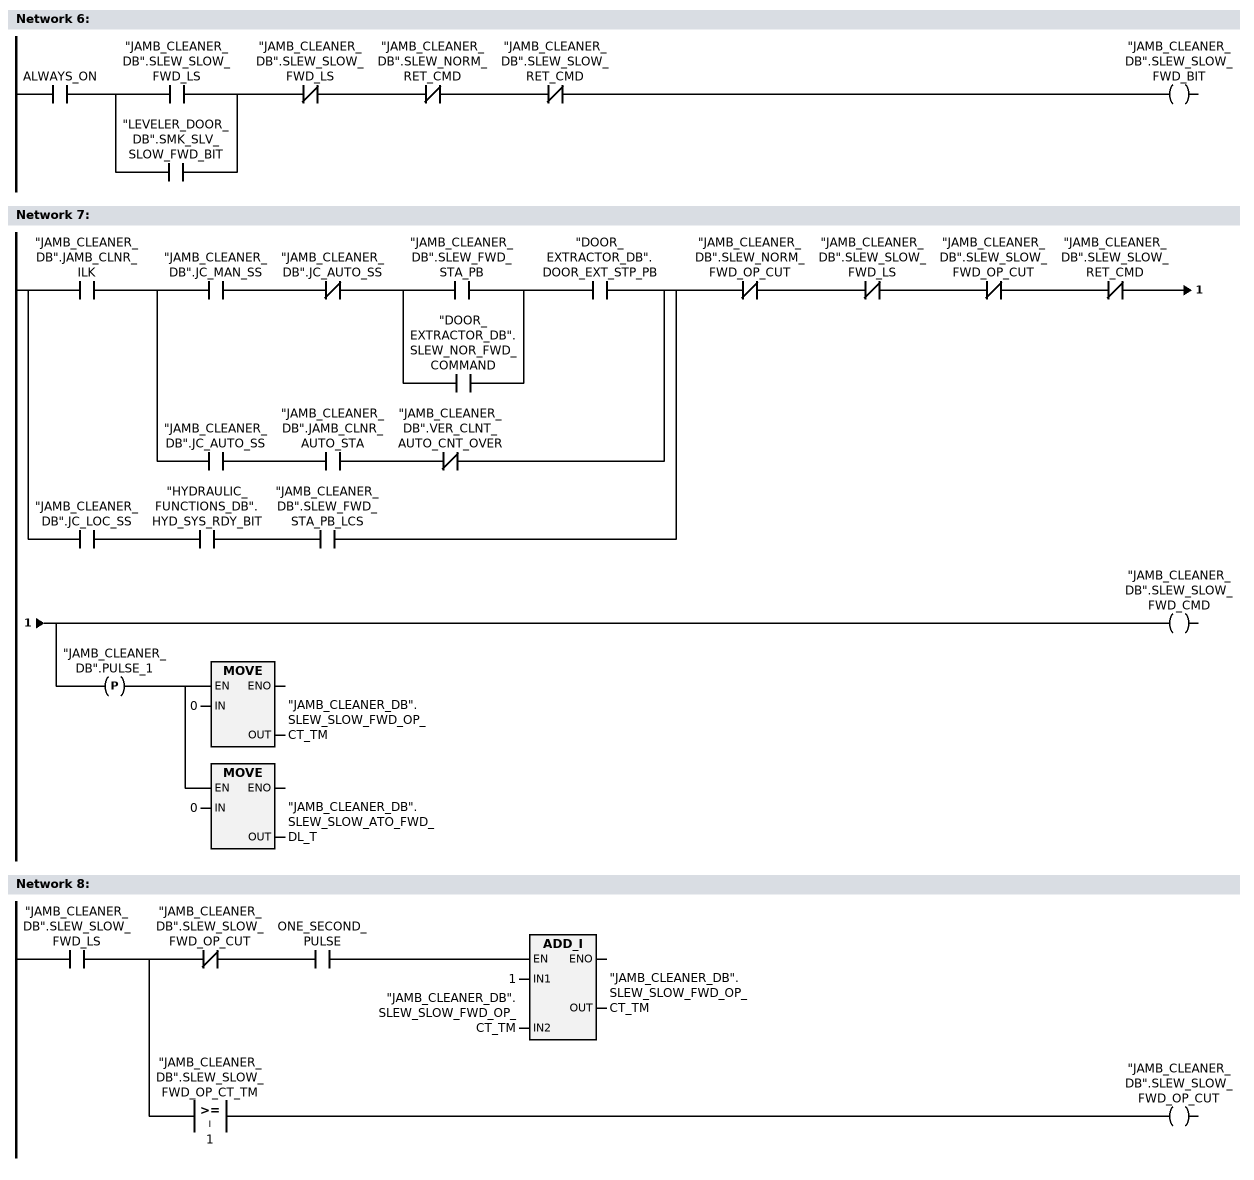
NETWORK
TITLE =
      A     "ALWAYS_ON";
      A(;
      O     "JAMB_CLEANER_DB".SLEW_SLOW_FWD_LS;
      O     "LEVELER_DOOR_DB".SMK_SLV_SLOW_FWD_BIT;
      );
      AN    "JAMB_CLEANER_DB".SLEW_SLOW_FWD_LS;
      AN    "JAMB_CLEANER_DB".SLEW_NORM_RET_CMD;
      AN    "JAMB_CLEANER_DB".SLEW_SLOW_RET_CMD;
      =     "JAMB_CLEANER_DB".SLEW_SLOW_FWD_BIT;
NETWORK
TITLE =
      A(;
      A     "JAMB_CLEANER_DB".JAMB_CLNR_ILK;
      A(;
      A     "JAMB_CLEANER_DB".JC_MAN_SS;
      AN    "JAMB_CLEANER_DB".JC_AUTO_SS;
      A(;
      O     "JAMB_CLEANER_DB".SLEW_FWD_STA_PB;
      O     "DOOR_EXTRACTOR_DB".SLEW_NOR_FWD_COMMAND;
      );
      A     "DOOR_EXTRACTOR_DB".DOOR_EXT_STP_PB;
      O;
      A     "JAMB_CLEANER_DB".JC_AUTO_SS;
      A     "JAMB_CLEANER_DB".JAMB_CLNR_AUTO_STA;
      AN    "JAMB_CLEANER_DB".VER_CLNT_AUTO_CNT_OVER;
      );
      O;
      A     "JAMB_CLEANER_DB".JC_LOC_SS;
      A     "HYDRAULIC_FUNCTIONS_DB".HYD_SYS_RDY_BIT;
      A     "JAMB_CLEANER_DB".SLEW_FWD_STA_PB_LCS;
      );
      AN    "JAMB_CLEANER_DB".SLEW_NORM_FWD_OP_CUT;
      AN    "JAMB_CLEANER_DB".SLEW_SLOW_FWD_LS;
      AN    "JAMB_CLEANER_DB".SLEW_SLOW_FWD_OP_CUT;
      AN    "JAMB_CLEANER_DB".SLEW_SLOW_RET_CMD;
      =     L 0.0;
      A     L 0.0;
      BLD   102;
      =     "JAMB_CLEANER_DB".SLEW_SLOW_FWD_CMD;
      A     L 0.0;
      FP    "JAMB_CLEANER_DB".PULSE_1;
      =     L 0.1;
      A     L 0.1;
      JNB   M002;
      L     0;
      T     "JAMB_CLEANER_DB".SLEW_SLOW_FWD_OP_CT_TM;
M002: NOP   0;
      A     L 0.1;
      JNB   M003;
      L     0;
      T     "JAMB_CLEANER_DB".SLEW_SLOW_ATO_FWD_DL_T;
M003: NOP   0;
NETWORK
TITLE =
      A     "JAMB_CLEANER_DB".SLEW_SLOW_FWD_LS;
      =     L 0.0;
      A     L 0.0;
      AN    "JAMB_CLEANER_DB".SLEW_SLOW_FWD_OP_CUT;
      A     "ONE_SECOND_PULSE";
      JNB   M004;
      L     1;
      L     "JAMB_CLEANER_DB".SLEW_SLOW_FWD_OP_CT_TM;
      +I;
      T     "JAMB_CLEANER_DB".SLEW_SLOW_FWD_OP_CT_TM;
M004: NOP   0;
      A     L 0.0;
      A(;
      L     "JAMB_CLEANER_DB".SLEW_SLOW_FWD_OP_CT_TM;
      L     1;
      >=I;
      );
      =     "JAMB_CLEANER_DB".SLEW_SLOW_FWD_OP_CUT;
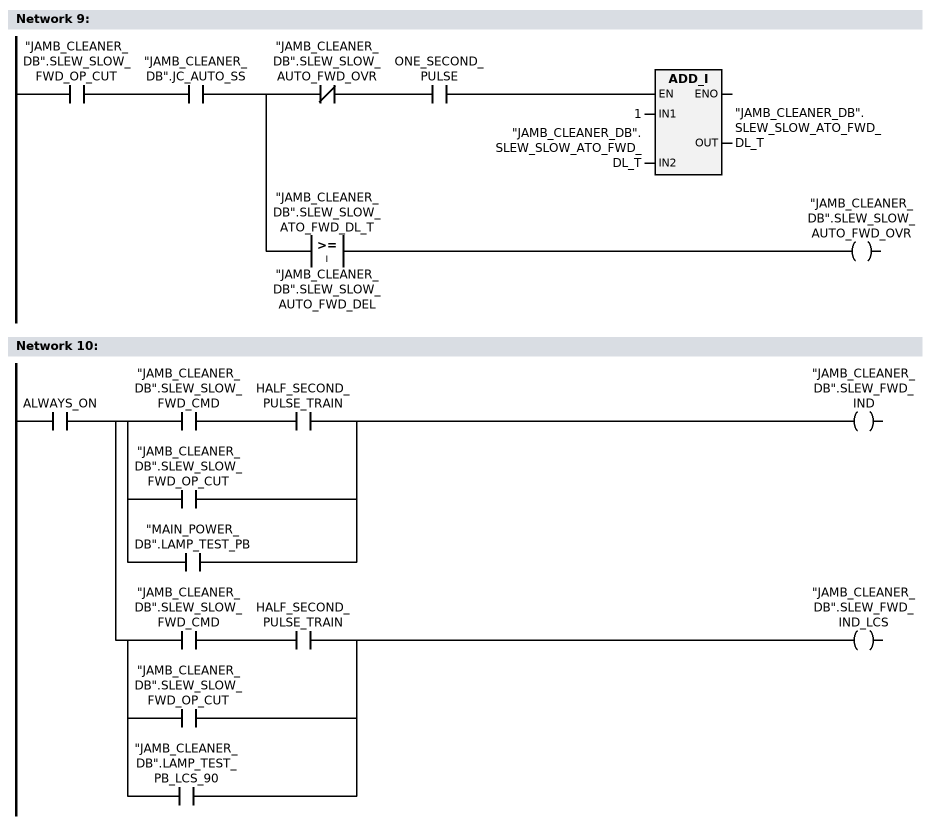
NETWORK
TITLE =
      A     "JAMB_CLEANER_DB".SLEW_SLOW_FWD_OP_CUT;
      A     "JAMB_CLEANER_DB".JC_AUTO_SS;
      =     L 0.0;
      A     L 0.0;
      AN    "JAMB_CLEANER_DB".SLEW_SLOW_AUTO_FWD_OVR;
      A     "ONE_SECOND_PULSE";
      JNB   M005;
      L     1;
      L     "JAMB_CLEANER_DB".SLEW_SLOW_ATO_FWD_DL_T;
      +I;
      T     "JAMB_CLEANER_DB".SLEW_SLOW_ATO_FWD_DL_T;
M005: NOP   0;
      A     L 0.0;
      A(;
      L     "JAMB_CLEANER_DB".SLEW_SLOW_ATO_FWD_DL_T;
      L     "JAMB_CLEANER_DB".SLEW_SLOW_AUTO_FWD_DEL;
      >=I;
      );
      =     "JAMB_CLEANER_DB".SLEW_SLOW_AUTO_FWD_OVR;
NETWORK
TITLE =
      A     "ALWAYS_ON";
      =     L 0.0;
      A     L 0.0;
      A(;
      A     "JAMB_CLEANER_DB".SLEW_SLOW_FWD_CMD;
      A     "HALF_SECOND_PULSE_TRAIN";
      O     "JAMB_CLEANER_DB".SLEW_SLOW_FWD_OP_CUT;
      O     "MAIN_POWER_DB".LAMP_TEST_PB;
      );
      =     "JAMB_CLEANER_DB".SLEW_FWD_IND;
      A     L 0.0;
      A(;
      A     "JAMB_CLEANER_DB".SLEW_SLOW_FWD_CMD;
      A     "HALF_SECOND_PULSE_TRAIN";
      O     "JAMB_CLEANER_DB".SLEW_SLOW_FWD_OP_CUT;
      O     "JAMB_CLEANER_DB".LAMP_TEST_PB_LCS_90;
      );
      =     "JAMB_CLEANER_DB".SLEW_FWD_IND_LCS;
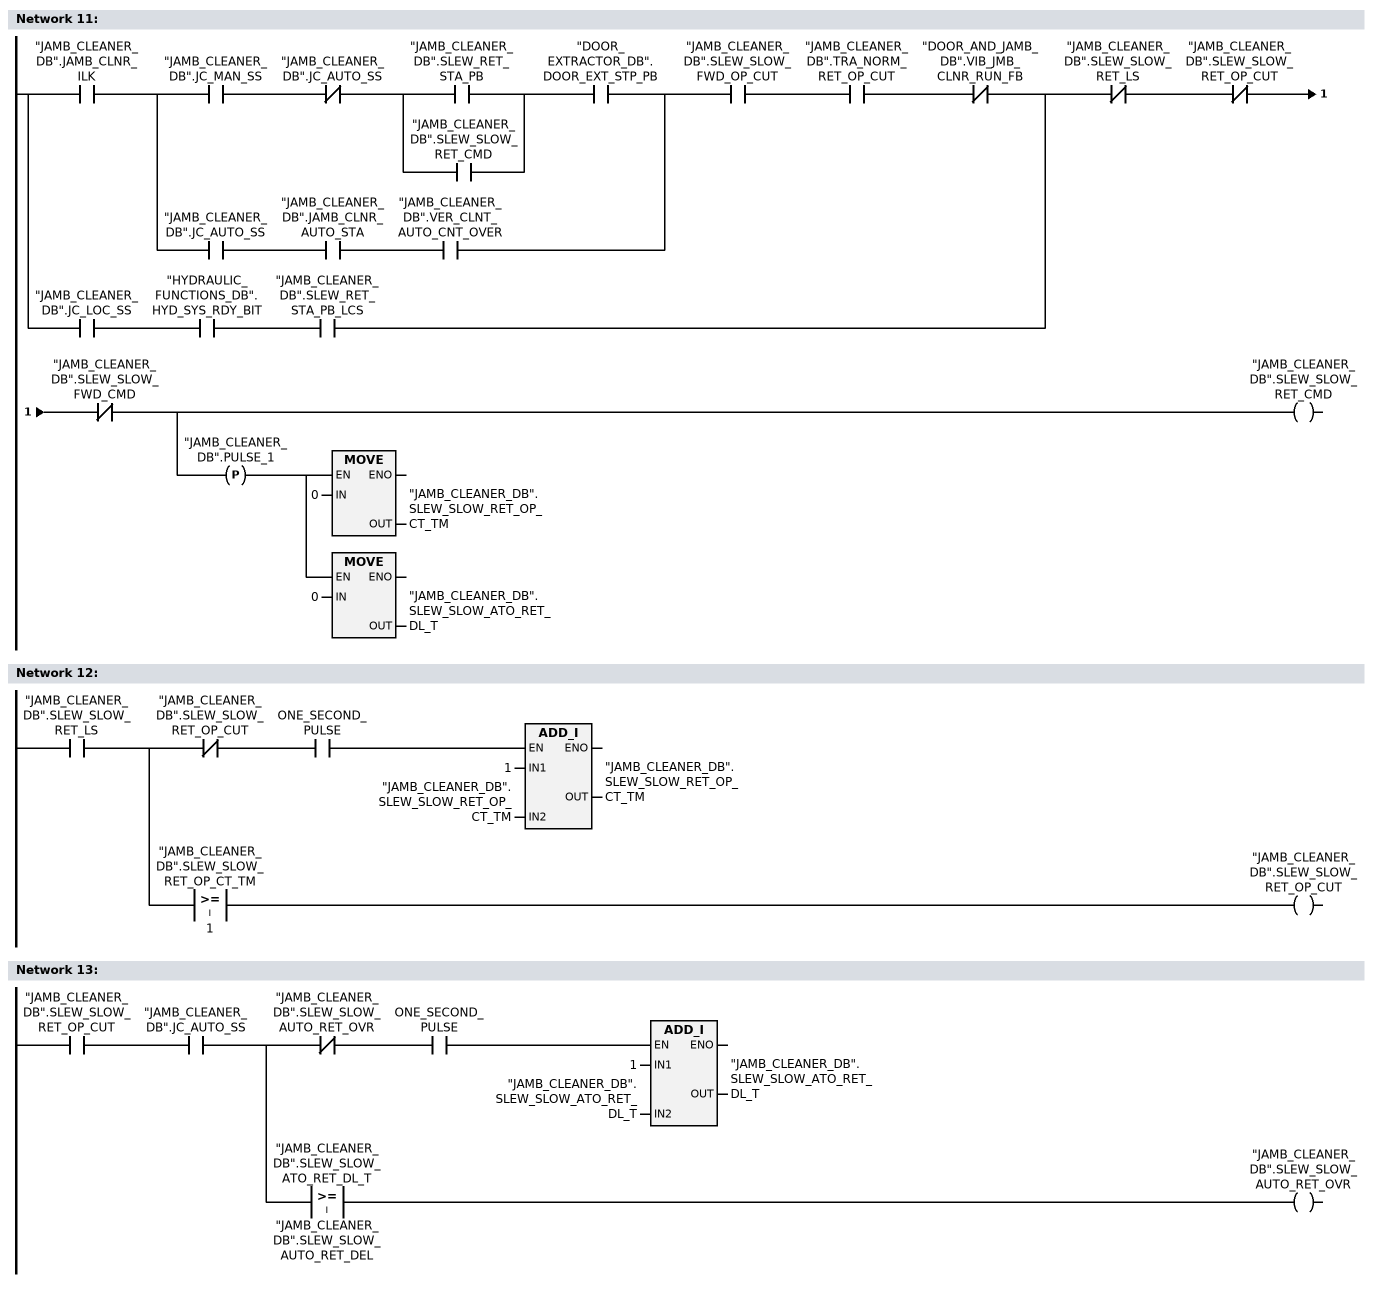
NETWORK
TITLE =
      A(;
      A     "JAMB_CLEANER_DB".JAMB_CLNR_ILK;
      A(;
      A     "JAMB_CLEANER_DB".JC_MAN_SS;
      AN    "JAMB_CLEANER_DB".JC_AUTO_SS;
      A(;
      O     "JAMB_CLEANER_DB".SLEW_RET_STA_PB;
      O     "JAMB_CLEANER_DB".SLEW_SLOW_RET_CMD;
      );
      A     "DOOR_EXTRACTOR_DB".DOOR_EXT_STP_PB;
      O;
      A     "JAMB_CLEANER_DB".JC_AUTO_SS;
      A     "JAMB_CLEANER_DB".JAMB_CLNR_AUTO_STA;
      A     "JAMB_CLEANER_DB".VER_CLNT_AUTO_CNT_OVER;
      );
      A     "JAMB_CLEANER_DB".SLEW_SLOW_FWD_OP_CUT;
      A     "JAMB_CLEANER_DB".TRA_NORM_RET_OP_CUT;
      AN    "DOOR_AND_JAMB_DB".VIB_JMB_CLNR_RUN_FB;
      O;
      A     "JAMB_CLEANER_DB".JC_LOC_SS;
      A     "HYDRAULIC_FUNCTIONS_DB".HYD_SYS_RDY_BIT;
      A     "JAMB_CLEANER_DB".SLEW_RET_STA_PB_LCS;
      );
      AN    "JAMB_CLEANER_DB".SLEW_SLOW_RET_LS;
      AN    "JAMB_CLEANER_DB".SLEW_SLOW_RET_OP_CUT;
      AN    "JAMB_CLEANER_DB".SLEW_SLOW_FWD_CMD;
      =     L 0.0;
      A     L 0.0;
      BLD   102;
      =     "JAMB_CLEANER_DB".SLEW_SLOW_RET_CMD;
      A     L 0.0;
      FP    "JAMB_CLEANER_DB".PULSE_1;
      =     L 0.1;
      A     L 0.1;
      JNB   M006;
      L     0;
      T     "JAMB_CLEANER_DB".SLEW_SLOW_RET_OP_CT_TM;
M006: NOP   0;
      A     L 0.1;
      JNB   M007;
      L     0;
      T     "JAMB_CLEANER_DB".SLEW_SLOW_ATO_RET_DL_T;
M007: NOP   0;
NETWORK
TITLE =
      A     "JAMB_CLEANER_DB".SLEW_SLOW_RET_LS;
      =     L 0.0;
      A     L 0.0;
      AN    "JAMB_CLEANER_DB".SLEW_SLOW_RET_OP_CUT;
      A     "ONE_SECOND_PULSE";
      JNB   M008;
      L     1;
      L     "JAMB_CLEANER_DB".SLEW_SLOW_RET_OP_CT_TM;
      +I;
      T     "JAMB_CLEANER_DB".SLEW_SLOW_RET_OP_CT_TM;
M008: NOP   0;
      A     L 0.0;
      A(;
      L     "JAMB_CLEANER_DB".SLEW_SLOW_RET_OP_CT_TM;
      L     1;
      >=I;
      );
      =     "JAMB_CLEANER_DB".SLEW_SLOW_RET_OP_CUT;
NETWORK
TITLE =
      A     "JAMB_CLEANER_DB".SLEW_SLOW_RET_OP_CUT;
      A     "JAMB_CLEANER_DB".JC_AUTO_SS;
      =     L 0.0;
      A     L 0.0;
      AN    "JAMB_CLEANER_DB".SLEW_SLOW_AUTO_RET_OVR;
      A     "ONE_SECOND_PULSE";
      JNB   M009;
      L     1;
      L     "JAMB_CLEANER_DB".SLEW_SLOW_ATO_RET_DL_T;
      +I;
      T     "JAMB_CLEANER_DB".SLEW_SLOW_ATO_RET_DL_T;
M009: NOP   0;
      A     L 0.0;
      A(;
      L     "JAMB_CLEANER_DB".SLEW_SLOW_ATO_RET_DL_T;
      L     "JAMB_CLEANER_DB".SLEW_SLOW_AUTO_RET_DEL;
      >=I;
      );
      =     "JAMB_CLEANER_DB".SLEW_SLOW_AUTO_RET_OVR;
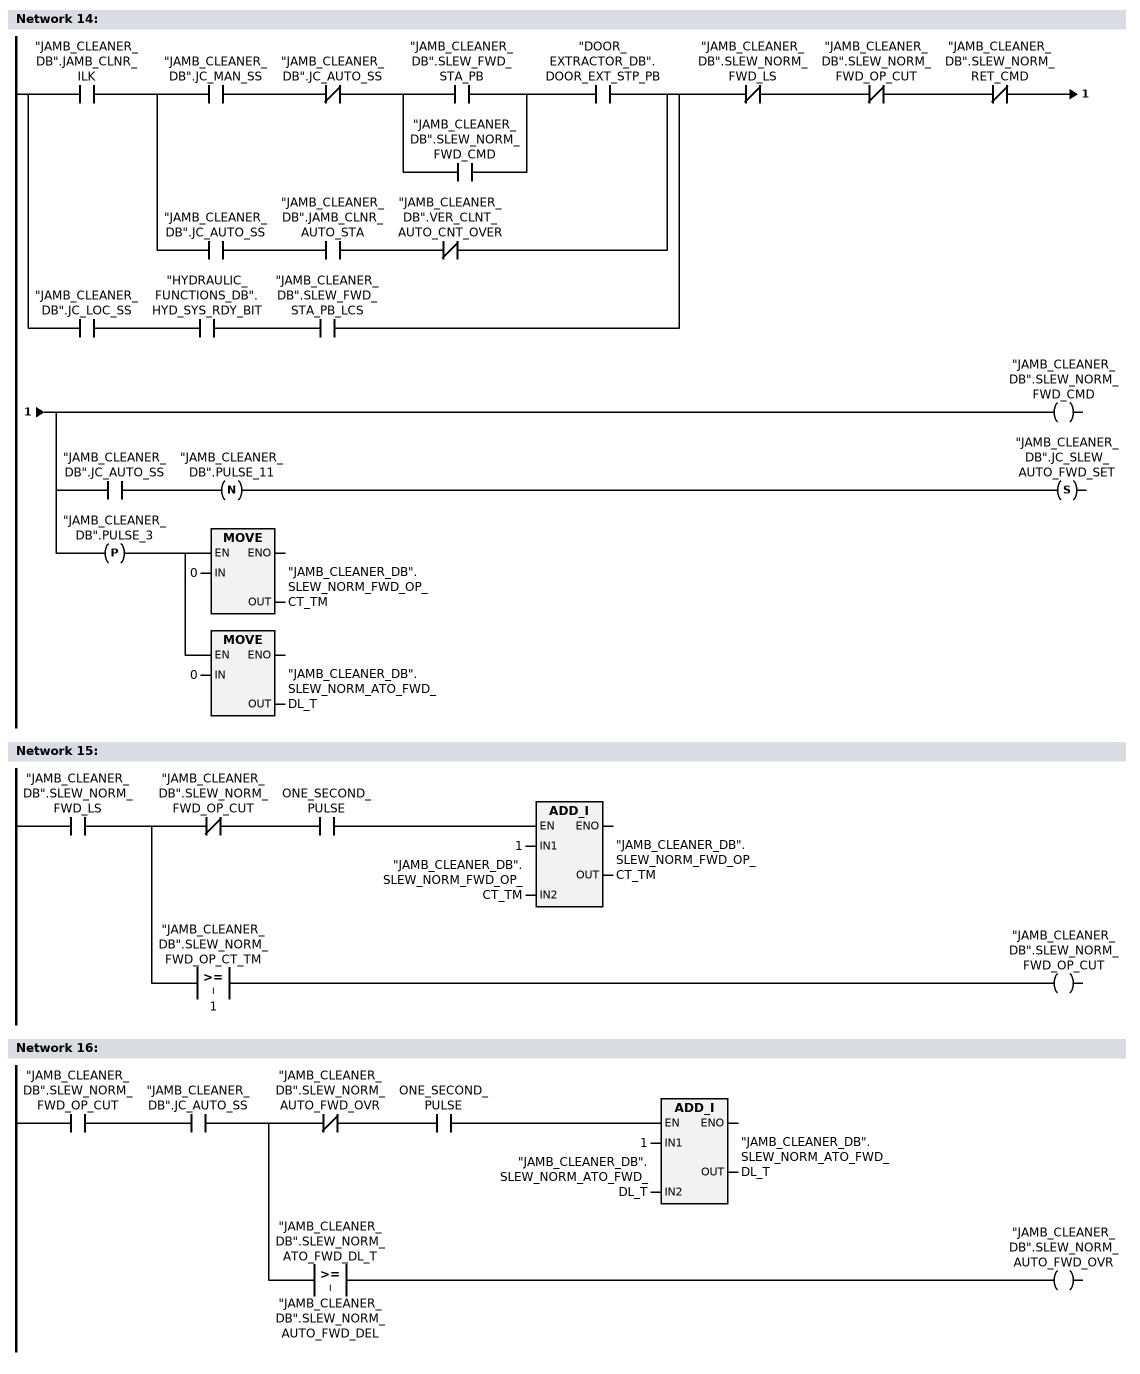
NETWORK
TITLE =
      A(;
      A     "JAMB_CLEANER_DB".JAMB_CLNR_ILK;
      A(;
      A     "JAMB_CLEANER_DB".JC_MAN_SS;
      AN    "JAMB_CLEANER_DB".JC_AUTO_SS;
      A(;
      O     "JAMB_CLEANER_DB".SLEW_FWD_STA_PB;
      O     "JAMB_CLEANER_DB".SLEW_NORM_FWD_CMD;
      );
      A     "DOOR_EXTRACTOR_DB".DOOR_EXT_STP_PB;
      O;
      A     "JAMB_CLEANER_DB".JC_AUTO_SS;
      A     "JAMB_CLEANER_DB".JAMB_CLNR_AUTO_STA;
      AN    "JAMB_CLEANER_DB".VER_CLNT_AUTO_CNT_OVER;
      );
      O;
      A     "JAMB_CLEANER_DB".JC_LOC_SS;
      A     "HYDRAULIC_FUNCTIONS_DB".HYD_SYS_RDY_BIT;
      A     "JAMB_CLEANER_DB".SLEW_FWD_STA_PB_LCS;
      );
      AN    "JAMB_CLEANER_DB".SLEW_NORM_FWD_LS;
      AN    "JAMB_CLEANER_DB".SLEW_NORM_FWD_OP_CUT;
      AN    "JAMB_CLEANER_DB".SLEW_NORM_RET_CMD;
      =     L 0.0;
      A     L 0.0;
      BLD   102;
      =     "JAMB_CLEANER_DB".SLEW_NORM_FWD_CMD;
      A     L 0.0;
      A     "JAMB_CLEANER_DB".JC_AUTO_SS;
      FN    "JAMB_CLEANER_DB".PULSE_11;
      S     "JAMB_CLEANER_DB".JC_SLEW_AUTO_FWD_SET;
      A     L 0.0;
      FP    "JAMB_CLEANER_DB".PULSE_3;
      =     L 0.1;
      A     L 0.1;
      JNB   M010;
      L     0;
      T     "JAMB_CLEANER_DB".SLEW_NORM_FWD_OP_CT_TM;
M010: NOP   0;
      A     L 0.1;
      JNB   M011;
      L     0;
      T     "JAMB_CLEANER_DB".SLEW_NORM_ATO_FWD_DL_T;
M011: NOP   0;
NETWORK
TITLE =
      A     "JAMB_CLEANER_DB".SLEW_NORM_FWD_LS;
      =     L 0.0;
      A     L 0.0;
      AN    "JAMB_CLEANER_DB".SLEW_NORM_FWD_OP_CUT;
      A     "ONE_SECOND_PULSE";
      JNB   M012;
      L     1;
      L     "JAMB_CLEANER_DB".SLEW_NORM_FWD_OP_CT_TM;
      +I;
      T     "JAMB_CLEANER_DB".SLEW_NORM_FWD_OP_CT_TM;
M012: NOP   0;
      A     L 0.0;
      A(;
      L     "JAMB_CLEANER_DB".SLEW_NORM_FWD_OP_CT_TM;
      L     1;
      >=I;
      );
      =     "JAMB_CLEANER_DB".SLEW_NORM_FWD_OP_CUT;
NETWORK
TITLE =
      A     "JAMB_CLEANER_DB".SLEW_NORM_FWD_OP_CUT;
      A     "JAMB_CLEANER_DB".JC_AUTO_SS;
      =     L 0.0;
      A     L 0.0;
      AN    "JAMB_CLEANER_DB".SLEW_NORM_AUTO_FWD_OVR;
      A     "ONE_SECOND_PULSE";
      JNB   M013;
      L     1;
      L     "JAMB_CLEANER_DB".SLEW_NORM_ATO_FWD_DL_T;
      +I;
      T     "JAMB_CLEANER_DB".SLEW_NORM_ATO_FWD_DL_T;
M013: NOP   0;
      A     L 0.0;
      A(;
      L     "JAMB_CLEANER_DB".SLEW_NORM_ATO_FWD_DL_T;
      L     "JAMB_CLEANER_DB".SLEW_NORM_AUTO_FWD_DEL;
      >=I;
      );
      =     "JAMB_CLEANER_DB".SLEW_NORM_AUTO_FWD_OVR;
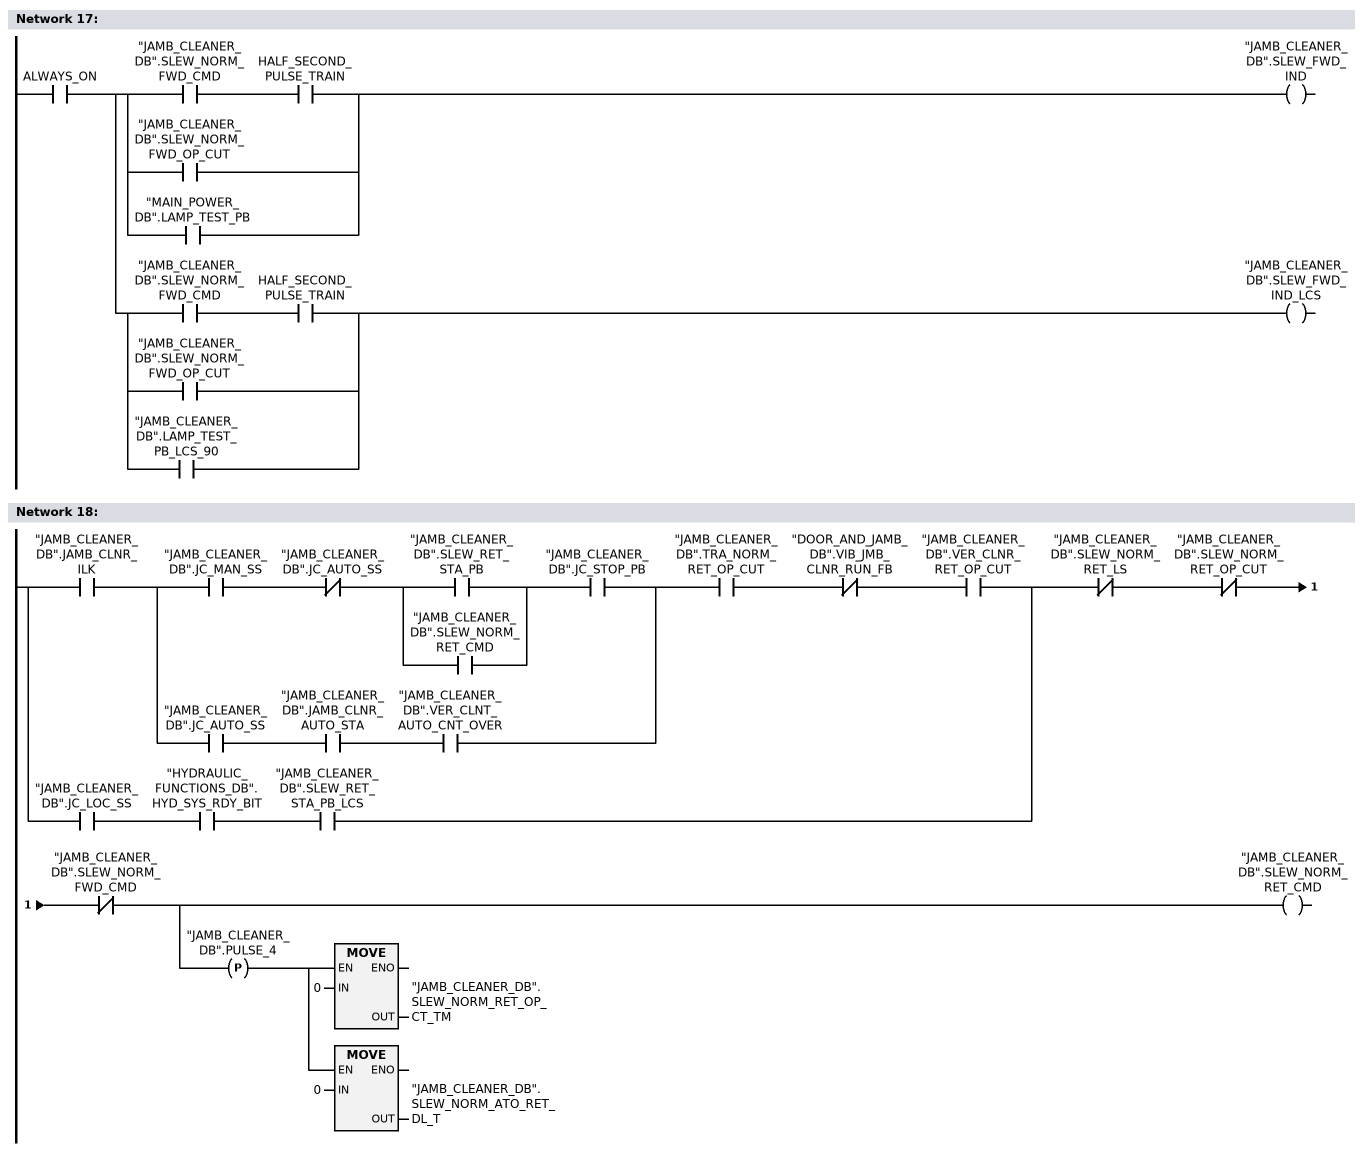
NETWORK
TITLE =
      A     "ALWAYS_ON";
      =     L 0.0;
      A     L 0.0;
      A(;
      A     "JAMB_CLEANER_DB".SLEW_NORM_FWD_CMD;
      A     "HALF_SECOND_PULSE_TRAIN";
      O     "JAMB_CLEANER_DB".SLEW_NORM_FWD_OP_CUT;
      O     "MAIN_POWER_DB".LAMP_TEST_PB;
      );
      =     "JAMB_CLEANER_DB".SLEW_FWD_IND;
      A     L 0.0;
      A(;
      A     "JAMB_CLEANER_DB".SLEW_NORM_FWD_CMD;
      A     "HALF_SECOND_PULSE_TRAIN";
      O     "JAMB_CLEANER_DB".SLEW_NORM_FWD_OP_CUT;
      O     "JAMB_CLEANER_DB".LAMP_TEST_PB_LCS_90;
      );
      =     "JAMB_CLEANER_DB".SLEW_FWD_IND_LCS;
NETWORK
TITLE =
      A(;
      A     "JAMB_CLEANER_DB".JAMB_CLNR_ILK;
      A(;
      A     "JAMB_CLEANER_DB".JC_MAN_SS;
      AN    "JAMB_CLEANER_DB".JC_AUTO_SS;
      A(;
      O     "JAMB_CLEANER_DB".SLEW_RET_STA_PB;
      O     "JAMB_CLEANER_DB".SLEW_NORM_RET_CMD;
      );
      A     "JAMB_CLEANER_DB".JC_STOP_PB;
      O;
      A     "JAMB_CLEANER_DB".JC_AUTO_SS;
      A     "JAMB_CLEANER_DB".JAMB_CLNR_AUTO_STA;
      A     "JAMB_CLEANER_DB".VER_CLNT_AUTO_CNT_OVER;
      );
      A     "JAMB_CLEANER_DB".TRA_NORM_RET_OP_CUT;
      AN    "DOOR_AND_JAMB_DB".VIB_JMB_CLNR_RUN_FB;
      A     "JAMB_CLEANER_DB".VER_CLNR_RET_OP_CUT;
      O;
      A     "JAMB_CLEANER_DB".JC_LOC_SS;
      A     "HYDRAULIC_FUNCTIONS_DB".HYD_SYS_RDY_BIT;
      A     "JAMB_CLEANER_DB".SLEW_RET_STA_PB_LCS;
      );
      AN    "JAMB_CLEANER_DB".SLEW_NORM_RET_LS;
      AN    "JAMB_CLEANER_DB".SLEW_NORM_RET_OP_CUT;
      AN    "JAMB_CLEANER_DB".SLEW_NORM_FWD_CMD;
      =     L 0.0;
      A     L 0.0;
      BLD   102;
      =     "JAMB_CLEANER_DB".SLEW_NORM_RET_CMD;
      A     L 0.0;
      FP    "JAMB_CLEANER_DB".PULSE_4;
      =     L 0.1;
      A     L 0.1;
      JNB   M014;
      L     0;
      T     "JAMB_CLEANER_DB".SLEW_NORM_RET_OP_CT_TM;
M014: NOP   0;
      A     L 0.1;
      JNB   M015;
      L     0;
      T     "JAMB_CLEANER_DB".SLEW_NORM_ATO_RET_DL_T;
M015: NOP   0;
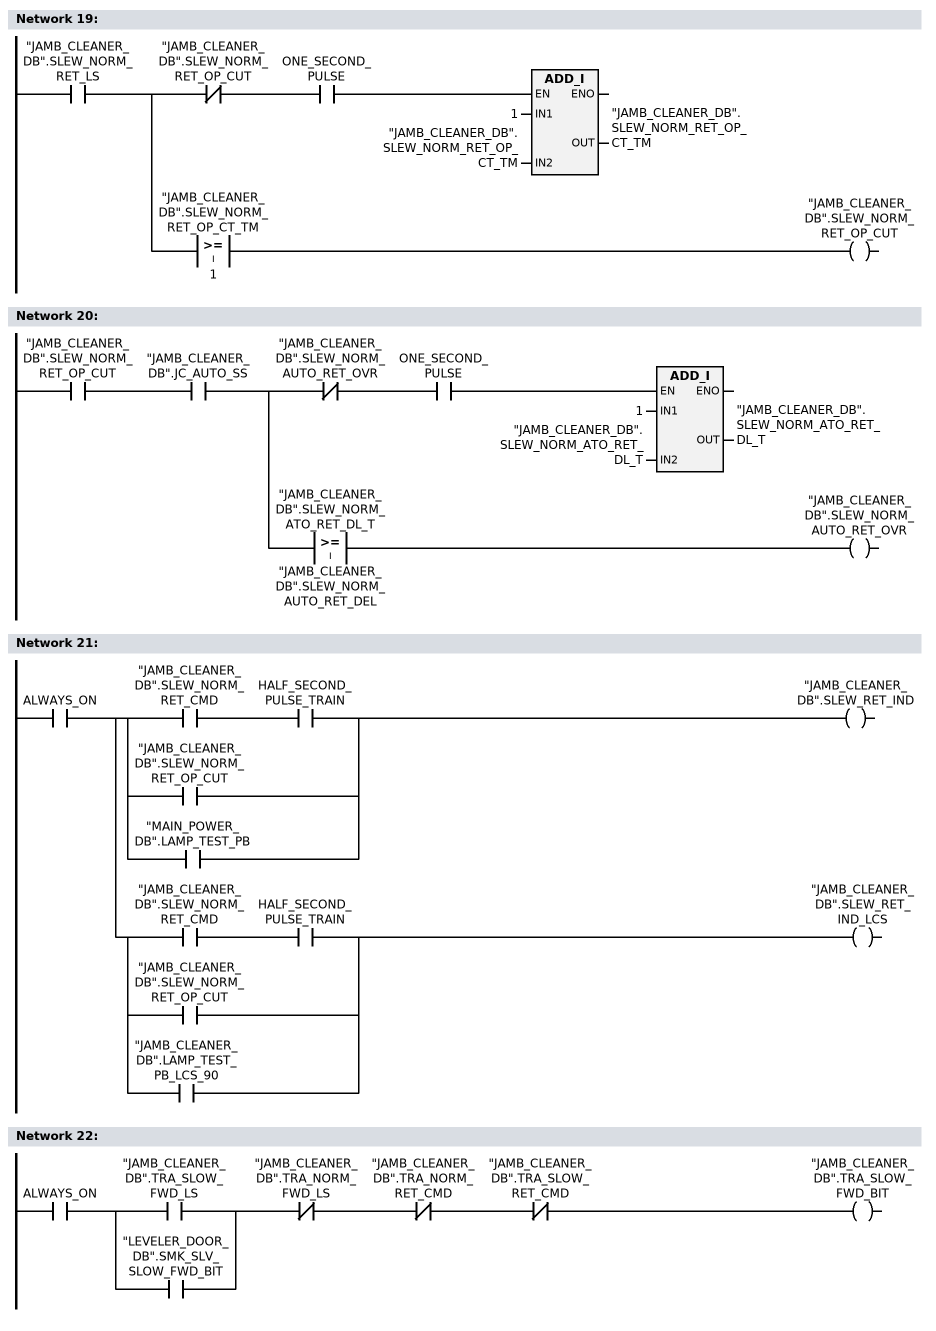
NETWORK
TITLE =
      A     "JAMB_CLEANER_DB".SLEW_NORM_RET_LS;
      =     L 0.0;
      A     L 0.0;
      AN    "JAMB_CLEANER_DB".SLEW_NORM_RET_OP_CUT;
      A     "ONE_SECOND_PULSE";
      JNB   M016;
      L     1;
      L     "JAMB_CLEANER_DB".SLEW_NORM_RET_OP_CT_TM;
      +I;
      T     "JAMB_CLEANER_DB".SLEW_NORM_RET_OP_CT_TM;
M016: NOP   0;
      A     L 0.0;
      A(;
      L     "JAMB_CLEANER_DB".SLEW_NORM_RET_OP_CT_TM;
      L     1;
      >=I;
      );
      =     "JAMB_CLEANER_DB".SLEW_NORM_RET_OP_CUT;
NETWORK
TITLE =
      A     "JAMB_CLEANER_DB".SLEW_NORM_RET_OP_CUT;
      A     "JAMB_CLEANER_DB".JC_AUTO_SS;
      =     L 0.0;
      A     L 0.0;
      AN    "JAMB_CLEANER_DB".SLEW_NORM_AUTO_RET_OVR;
      A     "ONE_SECOND_PULSE";
      JNB   M017;
      L     1;
      L     "JAMB_CLEANER_DB".SLEW_NORM_ATO_RET_DL_T;
      +I;
      T     "JAMB_CLEANER_DB".SLEW_NORM_ATO_RET_DL_T;
M017: NOP   0;
      A     L 0.0;
      A(;
      L     "JAMB_CLEANER_DB".SLEW_NORM_ATO_RET_DL_T;
      L     "JAMB_CLEANER_DB".SLEW_NORM_AUTO_RET_DEL;
      >=I;
      );
      =     "JAMB_CLEANER_DB".SLEW_NORM_AUTO_RET_OVR;
NETWORK
TITLE =
      A     "ALWAYS_ON";
      =     L 0.0;
      A     L 0.0;
      A(;
      A     "JAMB_CLEANER_DB".SLEW_NORM_RET_CMD;
      A     "HALF_SECOND_PULSE_TRAIN";
      O     "JAMB_CLEANER_DB".SLEW_NORM_RET_OP_CUT;
      O     "MAIN_POWER_DB".LAMP_TEST_PB;
      );
      =     "JAMB_CLEANER_DB".SLEW_RET_IND;
      A     L 0.0;
      A(;
      A     "JAMB_CLEANER_DB".SLEW_NORM_RET_CMD;
      A     "HALF_SECOND_PULSE_TRAIN";
      O     "JAMB_CLEANER_DB".SLEW_NORM_RET_OP_CUT;
      O     "JAMB_CLEANER_DB".LAMP_TEST_PB_LCS_90;
      );
      =     "JAMB_CLEANER_DB".SLEW_RET_IND_LCS;
NETWORK
TITLE =
      A     "ALWAYS_ON";
      A(;
      O     "JAMB_CLEANER_DB".TRA_SLOW_FWD_LS;
      O     "LEVELER_DOOR_DB".SMK_SLV_SLOW_FWD_BIT;
      );
      AN    "JAMB_CLEANER_DB".TRA_NORM_FWD_LS;
      AN    "JAMB_CLEANER_DB".TRA_NORM_RET_CMD;
      AN    "JAMB_CLEANER_DB".TRA_SLOW_RET_CMD;
      =     "JAMB_CLEANER_DB".TRA_SLOW_FWD_BIT;
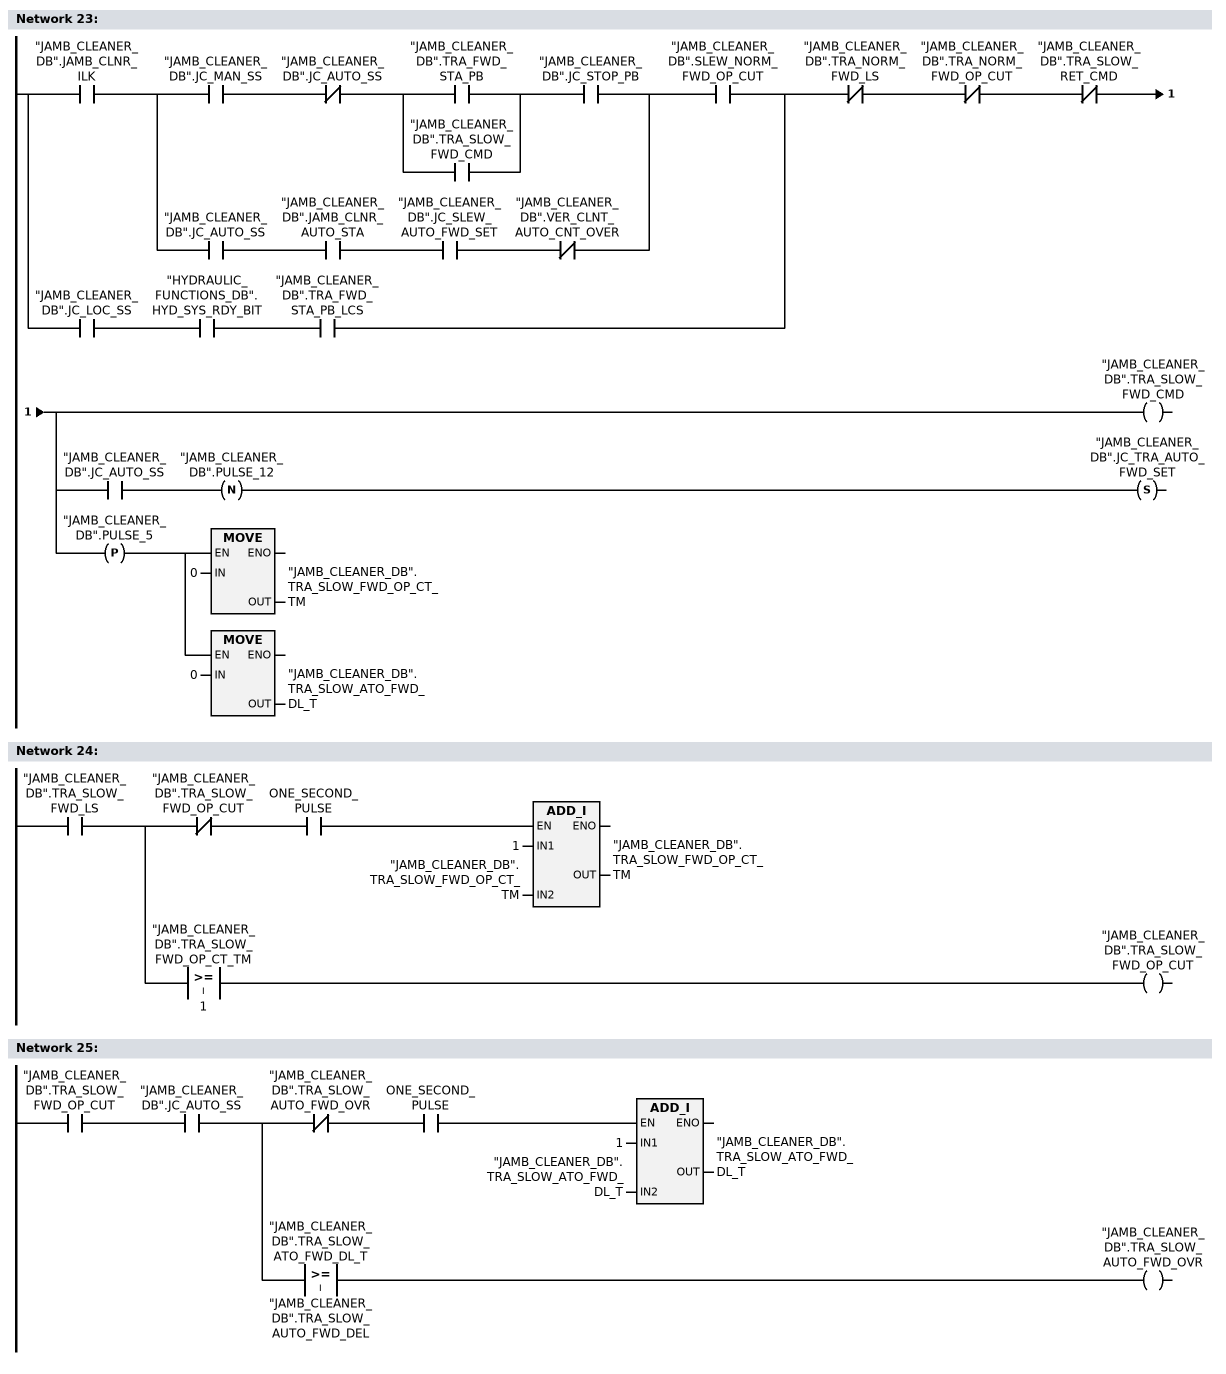
NETWORK
TITLE =
      A(;
      A     "JAMB_CLEANER_DB".JAMB_CLNR_ILK;
      A(;
      A     "JAMB_CLEANER_DB".JC_MAN_SS;
      AN    "JAMB_CLEANER_DB".JC_AUTO_SS;
      A(;
      O     "JAMB_CLEANER_DB".TRA_FWD_STA_PB;
      O     "JAMB_CLEANER_DB".TRA_SLOW_FWD_CMD;
      );
      A     "JAMB_CLEANER_DB".JC_STOP_PB;
      O;
      A     "JAMB_CLEANER_DB".JC_AUTO_SS;
      A     "JAMB_CLEANER_DB".JAMB_CLNR_AUTO_STA;
      A     "JAMB_CLEANER_DB".JC_SLEW_AUTO_FWD_SET;
      AN    "JAMB_CLEANER_DB".VER_CLNT_AUTO_CNT_OVER;
      );
      A     "JAMB_CLEANER_DB".SLEW_NORM_FWD_OP_CUT;
      O;
      A     "JAMB_CLEANER_DB".JC_LOC_SS;
      A     "HYDRAULIC_FUNCTIONS_DB".HYD_SYS_RDY_BIT;
      A     "JAMB_CLEANER_DB".TRA_FWD_STA_PB_LCS;
      );
      AN    "JAMB_CLEANER_DB".TRA_NORM_FWD_LS;
      AN    "JAMB_CLEANER_DB".TRA_NORM_FWD_OP_CUT;
      AN    "JAMB_CLEANER_DB".TRA_SLOW_RET_CMD;
      =     L 0.0;
      A     L 0.0;
      BLD   102;
      =     "JAMB_CLEANER_DB".TRA_SLOW_FWD_CMD;
      A     L 0.0;
      A     "JAMB_CLEANER_DB".JC_AUTO_SS;
      FN    "JAMB_CLEANER_DB".PULSE_12;
      S     "JAMB_CLEANER_DB".JC_TRA_AUTO_FWD_SET;
      A     L 0.0;
      FP    "JAMB_CLEANER_DB".PULSE_5;
      =     L 0.1;
      A     L 0.1;
      JNB   M018;
      L     0;
      T     "JAMB_CLEANER_DB".TRA_SLOW_FWD_OP_CT_TM;
M018: NOP   0;
      A     L 0.1;
      JNB   M019;
      L     0;
      T     "JAMB_CLEANER_DB".TRA_SLOW_ATO_FWD_DL_T;
M019: NOP   0;
NETWORK
TITLE =
      A     "JAMB_CLEANER_DB".TRA_SLOW_FWD_LS;
      =     L 0.0;
      A     L 0.0;
      AN    "JAMB_CLEANER_DB".TRA_SLOW_FWD_OP_CUT;
      A     "ONE_SECOND_PULSE";
      JNB   M020;
      L     1;
      L     "JAMB_CLEANER_DB".TRA_SLOW_FWD_OP_CT_TM;
      +I;
      T     "JAMB_CLEANER_DB".TRA_SLOW_FWD_OP_CT_TM;
M020: NOP   0;
      A     L 0.0;
      A(;
      L     "JAMB_CLEANER_DB".TRA_SLOW_FWD_OP_CT_TM;
      L     1;
      >=I;
      );
      =     "JAMB_CLEANER_DB".TRA_SLOW_FWD_OP_CUT;
NETWORK
TITLE =
      A     "JAMB_CLEANER_DB".TRA_SLOW_FWD_OP_CUT;
      A     "JAMB_CLEANER_DB".JC_AUTO_SS;
      =     L 0.0;
      A     L 0.0;
      AN    "JAMB_CLEANER_DB".TRA_SLOW_AUTO_FWD_OVR;
      A     "ONE_SECOND_PULSE";
      JNB   M021;
      L     1;
      L     "JAMB_CLEANER_DB".TRA_SLOW_ATO_FWD_DL_T;
      +I;
      T     "JAMB_CLEANER_DB".TRA_SLOW_ATO_FWD_DL_T;
M021: NOP   0;
      A     L 0.0;
      A(;
      L     "JAMB_CLEANER_DB".TRA_SLOW_ATO_FWD_DL_T;
      L     "JAMB_CLEANER_DB".TRA_SLOW_AUTO_FWD_DEL;
      >=I;
      );
      =     "JAMB_CLEANER_DB".TRA_SLOW_AUTO_FWD_OVR;
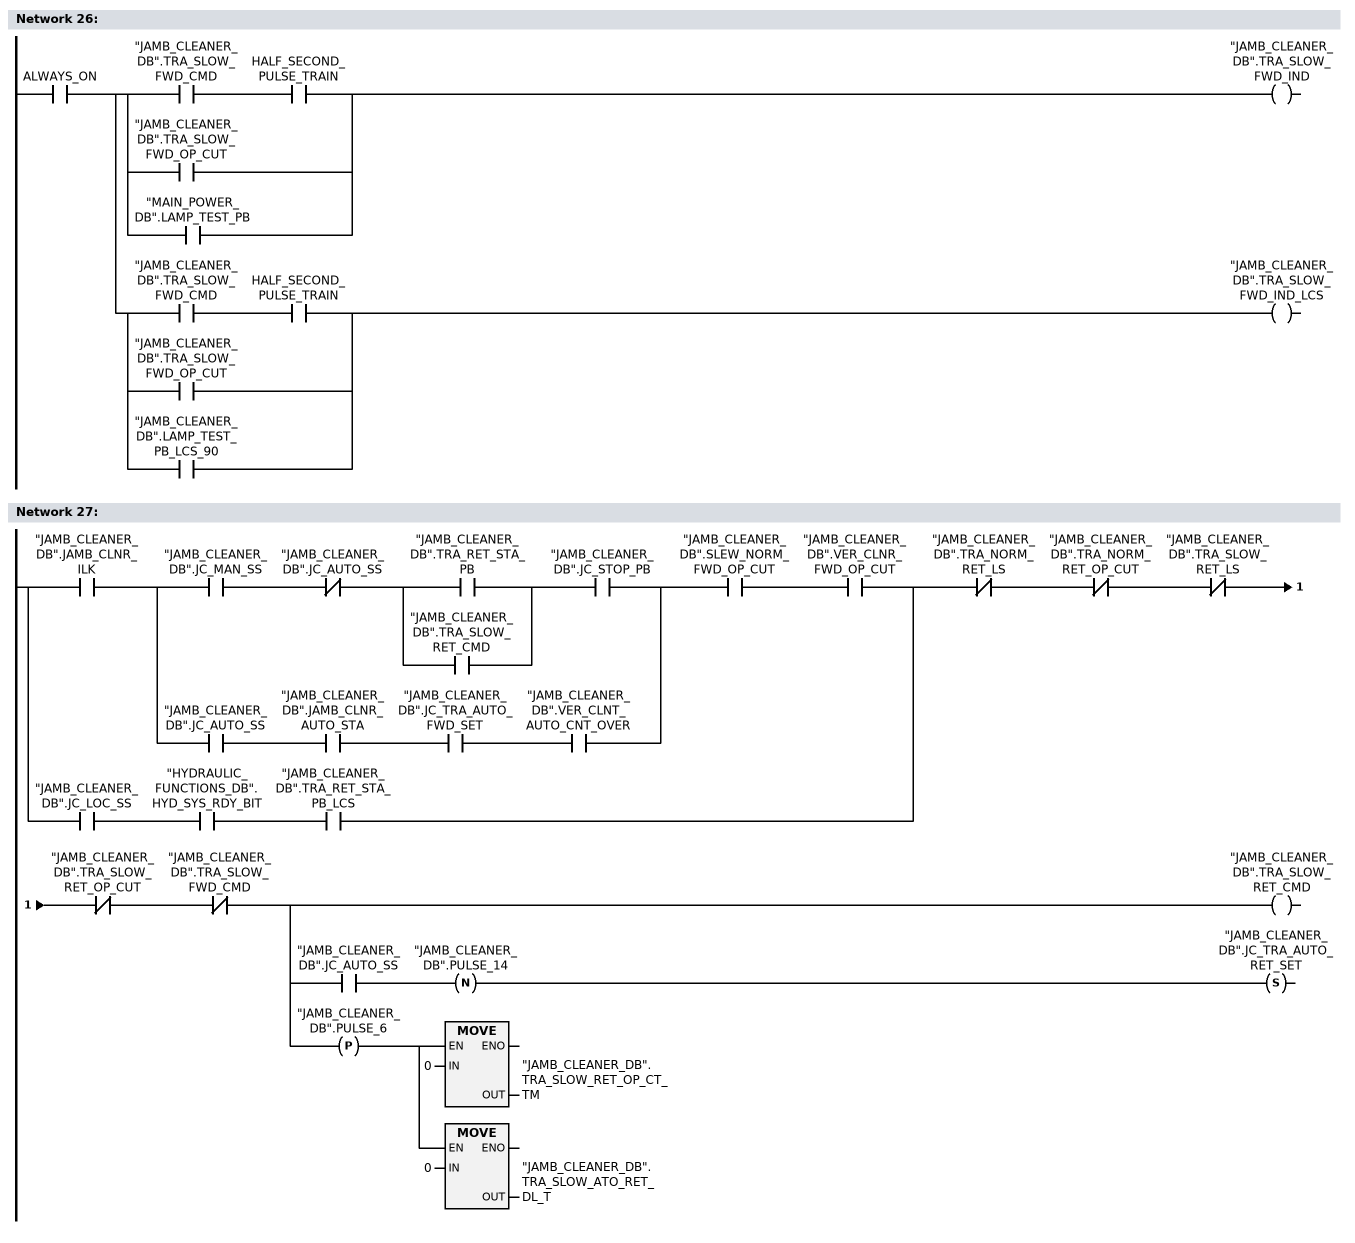
NETWORK
TITLE =
      A     "ALWAYS_ON";
      =     L 0.0;
      A     L 0.0;
      A(;
      A     "JAMB_CLEANER_DB".TRA_SLOW_FWD_CMD;
      A     "HALF_SECOND_PULSE_TRAIN";
      O     "JAMB_CLEANER_DB".TRA_SLOW_FWD_OP_CUT;
      O     "MAIN_POWER_DB".LAMP_TEST_PB;
      );
      =     "JAMB_CLEANER_DB".TRA_SLOW_FWD_IND;
      A     L 0.0;
      A(;
      A     "JAMB_CLEANER_DB".TRA_SLOW_FWD_CMD;
      A     "HALF_SECOND_PULSE_TRAIN";
      O     "JAMB_CLEANER_DB".TRA_SLOW_FWD_OP_CUT;
      O     "JAMB_CLEANER_DB".LAMP_TEST_PB_LCS_90;
      );
      =     "JAMB_CLEANER_DB".TRA_SLOW_FWD_IND_LCS;
NETWORK
TITLE =
      A(;
      A     "JAMB_CLEANER_DB".JAMB_CLNR_ILK;
      A(;
      A     "JAMB_CLEANER_DB".JC_MAN_SS;
      AN    "JAMB_CLEANER_DB".JC_AUTO_SS;
      A(;
      O     "JAMB_CLEANER_DB".TRA_RET_STA_PB;
      O     "JAMB_CLEANER_DB".TRA_SLOW_RET_CMD;
      );
      A     "JAMB_CLEANER_DB".JC_STOP_PB;
      O;
      A     "JAMB_CLEANER_DB".JC_AUTO_SS;
      A     "JAMB_CLEANER_DB".JAMB_CLNR_AUTO_STA;
      A     "JAMB_CLEANER_DB".JC_TRA_AUTO_FWD_SET;
      A     "JAMB_CLEANER_DB".VER_CLNT_AUTO_CNT_OVER;
      );
      A     "JAMB_CLEANER_DB".SLEW_NORM_FWD_OP_CUT;
      A     "JAMB_CLEANER_DB".VER_CLNR_FWD_OP_CUT;
      O;
      A     "JAMB_CLEANER_DB".JC_LOC_SS;
      A     "HYDRAULIC_FUNCTIONS_DB".HYD_SYS_RDY_BIT;
      A     "JAMB_CLEANER_DB".TRA_RET_STA_PB_LCS;
      );
      AN    "JAMB_CLEANER_DB".TRA_NORM_RET_LS;
      AN    "JAMB_CLEANER_DB".TRA_NORM_RET_OP_CUT;
      AN    "JAMB_CLEANER_DB".TRA_SLOW_RET_LS;
      AN    "JAMB_CLEANER_DB".TRA_SLOW_RET_OP_CUT;
      AN    "JAMB_CLEANER_DB".TRA_SLOW_FWD_CMD;
      =     L 0.0;
      A     L 0.0;
      BLD   102;
      =     "JAMB_CLEANER_DB".TRA_SLOW_RET_CMD;
      A     L 0.0;
      A     "JAMB_CLEANER_DB".JC_AUTO_SS;
      FN    "JAMB_CLEANER_DB".PULSE_14;
      S     "JAMB_CLEANER_DB".JC_TRA_AUTO_RET_SET;
      A     L 0.0;
      FP    "JAMB_CLEANER_DB".PULSE_6;
      =     L 0.1;
      A     L 0.1;
      JNB   M022;
      L     0;
      T     "JAMB_CLEANER_DB".TRA_SLOW_RET_OP_CT_TM;
M022: NOP   0;
      A     L 0.1;
      JNB   M023;
      L     0;
      T     "JAMB_CLEANER_DB".TRA_SLOW_ATO_RET_DL_T;
M023: NOP   0;
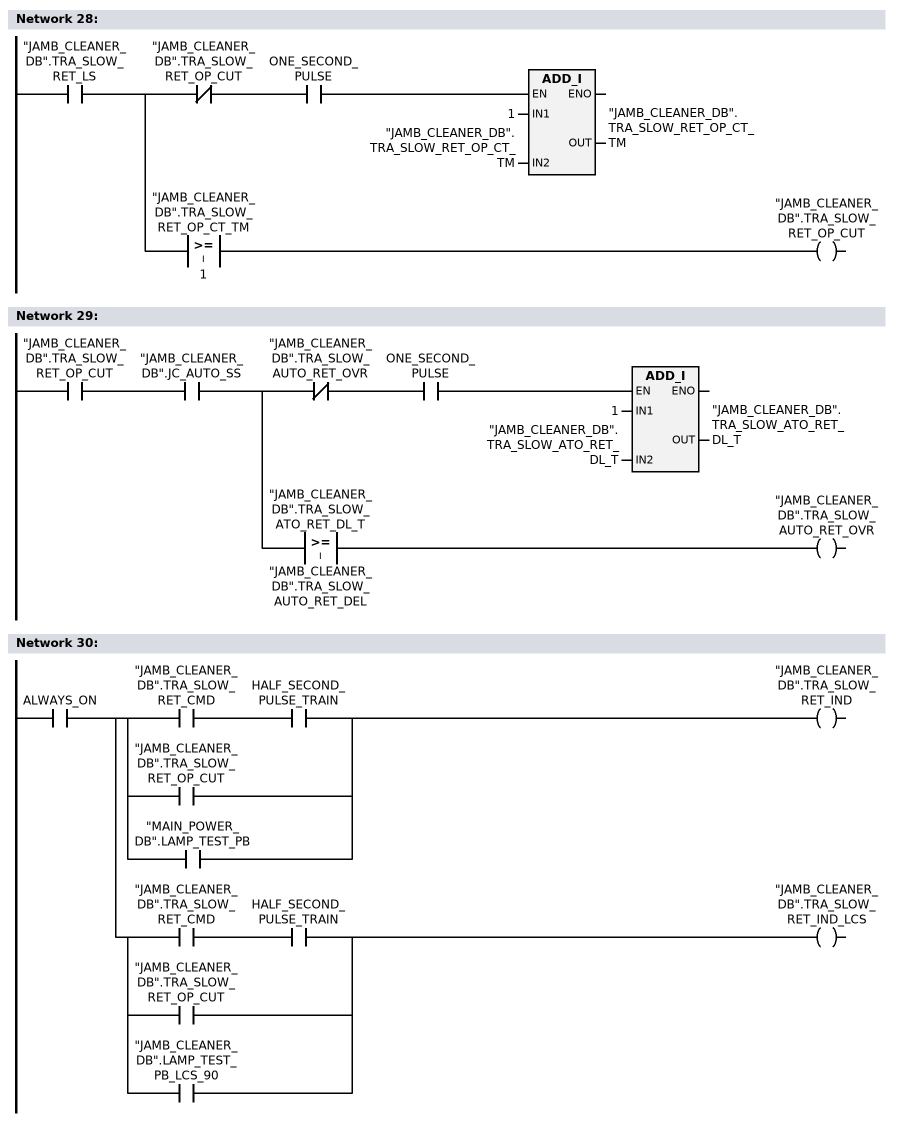
NETWORK
TITLE =
      A     "JAMB_CLEANER_DB".TRA_SLOW_RET_LS;
      =     L 0.0;
      A     L 0.0;
      AN    "JAMB_CLEANER_DB".TRA_SLOW_RET_OP_CUT;
      A     "ONE_SECOND_PULSE";
      JNB   M024;
      L     1;
      L     "JAMB_CLEANER_DB".TRA_SLOW_RET_OP_CT_TM;
      +I;
      T     "JAMB_CLEANER_DB".TRA_SLOW_RET_OP_CT_TM;
M024: NOP   0;
      A     L 0.0;
      A(;
      L     "JAMB_CLEANER_DB".TRA_SLOW_RET_OP_CT_TM;
      L     1;
      >=I;
      );
      =     "JAMB_CLEANER_DB".TRA_SLOW_RET_OP_CUT;
NETWORK
TITLE =
      A     "JAMB_CLEANER_DB".TRA_SLOW_RET_OP_CUT;
      A     "JAMB_CLEANER_DB".JC_AUTO_SS;
      =     L 0.0;
      A     L 0.0;
      AN    "JAMB_CLEANER_DB".TRA_SLOW_AUTO_RET_OVR;
      A     "ONE_SECOND_PULSE";
      JNB   M025;
      L     1;
      L     "JAMB_CLEANER_DB".TRA_SLOW_ATO_RET_DL_T;
      +I;
      T     "JAMB_CLEANER_DB".TRA_SLOW_ATO_RET_DL_T;
M025: NOP   0;
      A     L 0.0;
      A(;
      L     "JAMB_CLEANER_DB".TRA_SLOW_ATO_RET_DL_T;
      L     "JAMB_CLEANER_DB".TRA_SLOW_AUTO_RET_DEL;
      >=I;
      );
      =     "JAMB_CLEANER_DB".TRA_SLOW_AUTO_RET_OVR;
NETWORK
TITLE =
      A     "ALWAYS_ON";
      =     L 0.0;
      A     L 0.0;
      A(;
      A     "JAMB_CLEANER_DB".TRA_SLOW_RET_CMD;
      A     "HALF_SECOND_PULSE_TRAIN";
      O     "JAMB_CLEANER_DB".TRA_SLOW_RET_OP_CUT;
      O     "MAIN_POWER_DB".LAMP_TEST_PB;
      );
      =     "JAMB_CLEANER_DB".TRA_SLOW_RET_IND;
      A     L 0.0;
      A(;
      A     "JAMB_CLEANER_DB".TRA_SLOW_RET_CMD;
      A     "HALF_SECOND_PULSE_TRAIN";
      O     "JAMB_CLEANER_DB".TRA_SLOW_RET_OP_CUT;
      O     "JAMB_CLEANER_DB".LAMP_TEST_PB_LCS_90;
      );
      =     "JAMB_CLEANER_DB".TRA_SLOW_RET_IND_LCS;
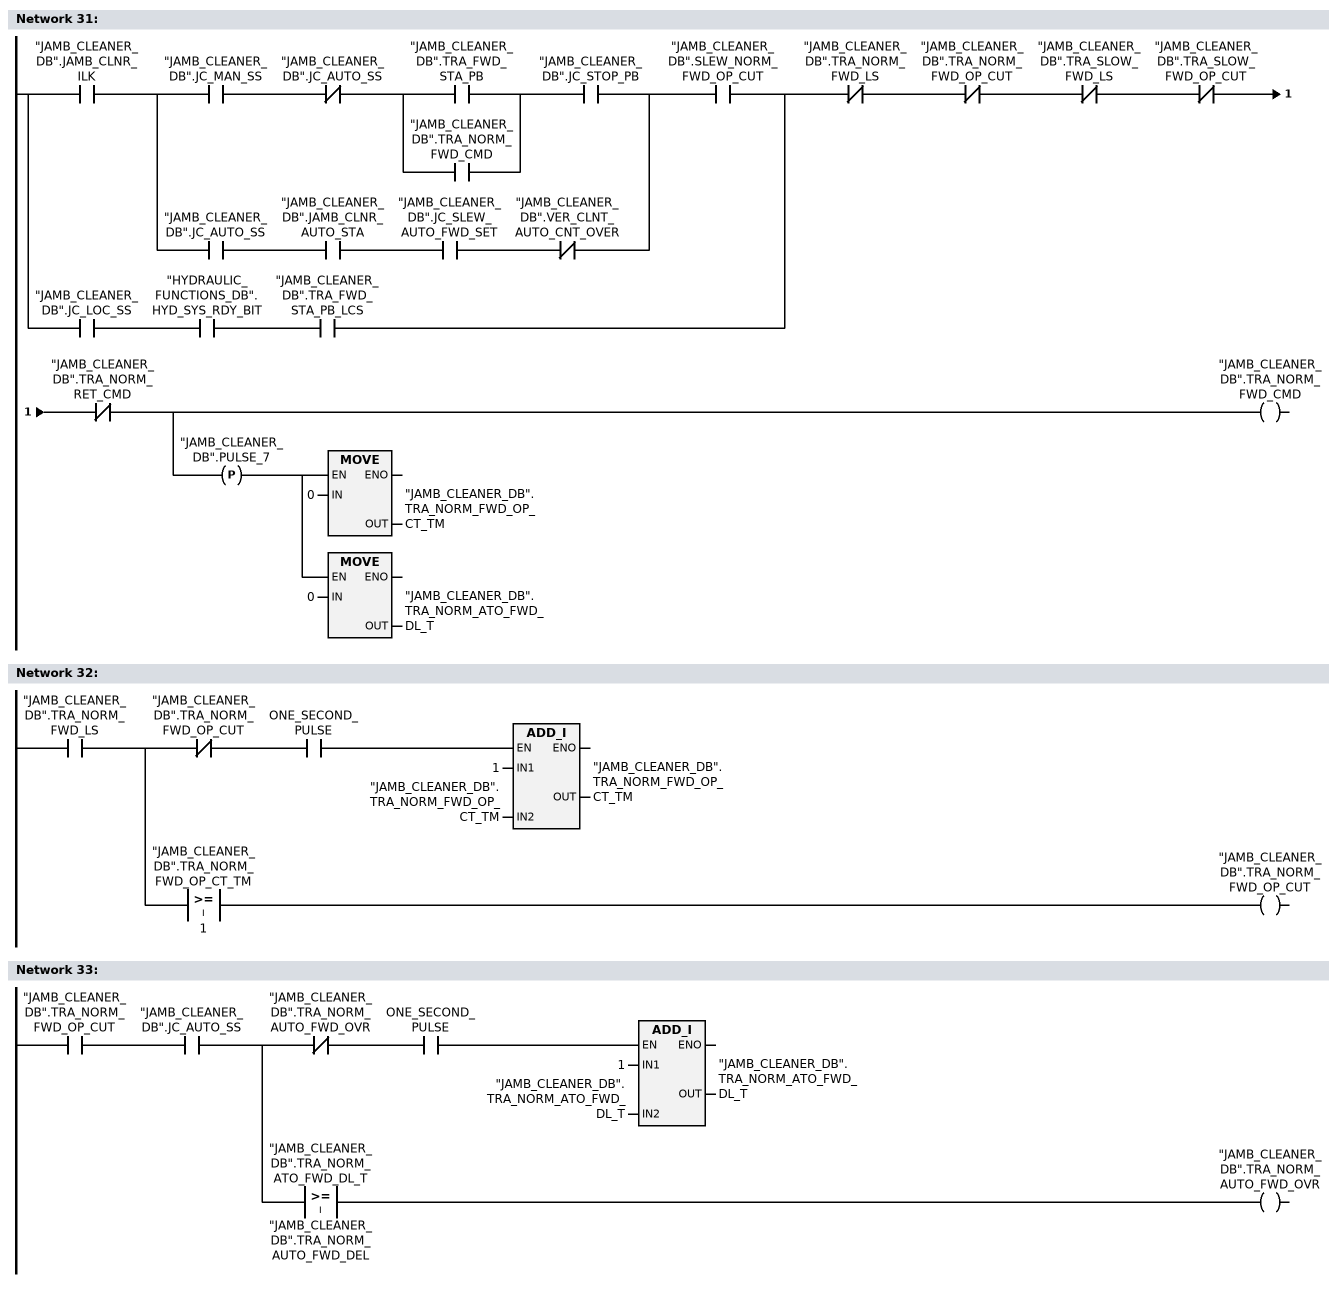
NETWORK
TITLE =
      A(;
      A     "JAMB_CLEANER_DB".JAMB_CLNR_ILK;
      A(;
      A     "JAMB_CLEANER_DB".JC_MAN_SS;
      AN    "JAMB_CLEANER_DB".JC_AUTO_SS;
      A(;
      O     "JAMB_CLEANER_DB".TRA_FWD_STA_PB;
      O     "JAMB_CLEANER_DB".TRA_NORM_FWD_CMD;
      );
      A     "JAMB_CLEANER_DB".JC_STOP_PB;
      O;
      A     "JAMB_CLEANER_DB".JC_AUTO_SS;
      A     "JAMB_CLEANER_DB".JAMB_CLNR_AUTO_STA;
      A     "JAMB_CLEANER_DB".JC_SLEW_AUTO_FWD_SET;
      AN    "JAMB_CLEANER_DB".VER_CLNT_AUTO_CNT_OVER;
      );
      A     "JAMB_CLEANER_DB".SLEW_NORM_FWD_OP_CUT;
      O;
      A     "JAMB_CLEANER_DB".JC_LOC_SS;
      A     "HYDRAULIC_FUNCTIONS_DB".HYD_SYS_RDY_BIT;
      A     "JAMB_CLEANER_DB".TRA_FWD_STA_PB_LCS;
      );
      AN    "JAMB_CLEANER_DB".TRA_NORM_FWD_LS;
      AN    "JAMB_CLEANER_DB".TRA_NORM_FWD_OP_CUT;
      AN    "JAMB_CLEANER_DB".TRA_SLOW_FWD_LS;
      AN    "JAMB_CLEANER_DB".TRA_SLOW_FWD_OP_CUT;
      AN    "JAMB_CLEANER_DB".TRA_NORM_RET_CMD;
      =     L 0.0;
      A     L 0.0;
      BLD   102;
      =     "JAMB_CLEANER_DB".TRA_NORM_FWD_CMD;
      A     L 0.0;
      FP    "JAMB_CLEANER_DB".PULSE_7;
      =     L 0.1;
      A     L 0.1;
      JNB   M026;
      L     0;
      T     "JAMB_CLEANER_DB".TRA_NORM_FWD_OP_CT_TM;
M026: NOP   0;
      A     L 0.1;
      JNB   M027;
      L     0;
      T     "JAMB_CLEANER_DB".TRA_NORM_ATO_FWD_DL_T;
M027: NOP   0;
NETWORK
TITLE =
      A     "JAMB_CLEANER_DB".TRA_NORM_FWD_LS;
      =     L 0.0;
      A     L 0.0;
      AN    "JAMB_CLEANER_DB".TRA_NORM_FWD_OP_CUT;
      A     "ONE_SECOND_PULSE";
      JNB   M028;
      L     1;
      L     "JAMB_CLEANER_DB".TRA_NORM_FWD_OP_CT_TM;
      +I;
      T     "JAMB_CLEANER_DB".TRA_NORM_FWD_OP_CT_TM;
M028: NOP   0;
      A     L 0.0;
      A(;
      L     "JAMB_CLEANER_DB".TRA_NORM_FWD_OP_CT_TM;
      L     1;
      >=I;
      );
      =     "JAMB_CLEANER_DB".TRA_NORM_FWD_OP_CUT;
NETWORK
TITLE =
      A     "JAMB_CLEANER_DB".TRA_NORM_FWD_OP_CUT;
      A     "JAMB_CLEANER_DB".JC_AUTO_SS;
      =     L 0.0;
      A     L 0.0;
      AN    "JAMB_CLEANER_DB".TRA_NORM_AUTO_FWD_OVR;
      A     "ONE_SECOND_PULSE";
      JNB   M029;
      L     1;
      L     "JAMB_CLEANER_DB".TRA_NORM_ATO_FWD_DL_T;
      +I;
      T     "JAMB_CLEANER_DB".TRA_NORM_ATO_FWD_DL_T;
M029: NOP   0;
      A     L 0.0;
      A(;
      L     "JAMB_CLEANER_DB".TRA_NORM_ATO_FWD_DL_T;
      L     "JAMB_CLEANER_DB".TRA_NORM_AUTO_FWD_DEL;
      >=I;
      );
      =     "JAMB_CLEANER_DB".TRA_NORM_AUTO_FWD_OVR;
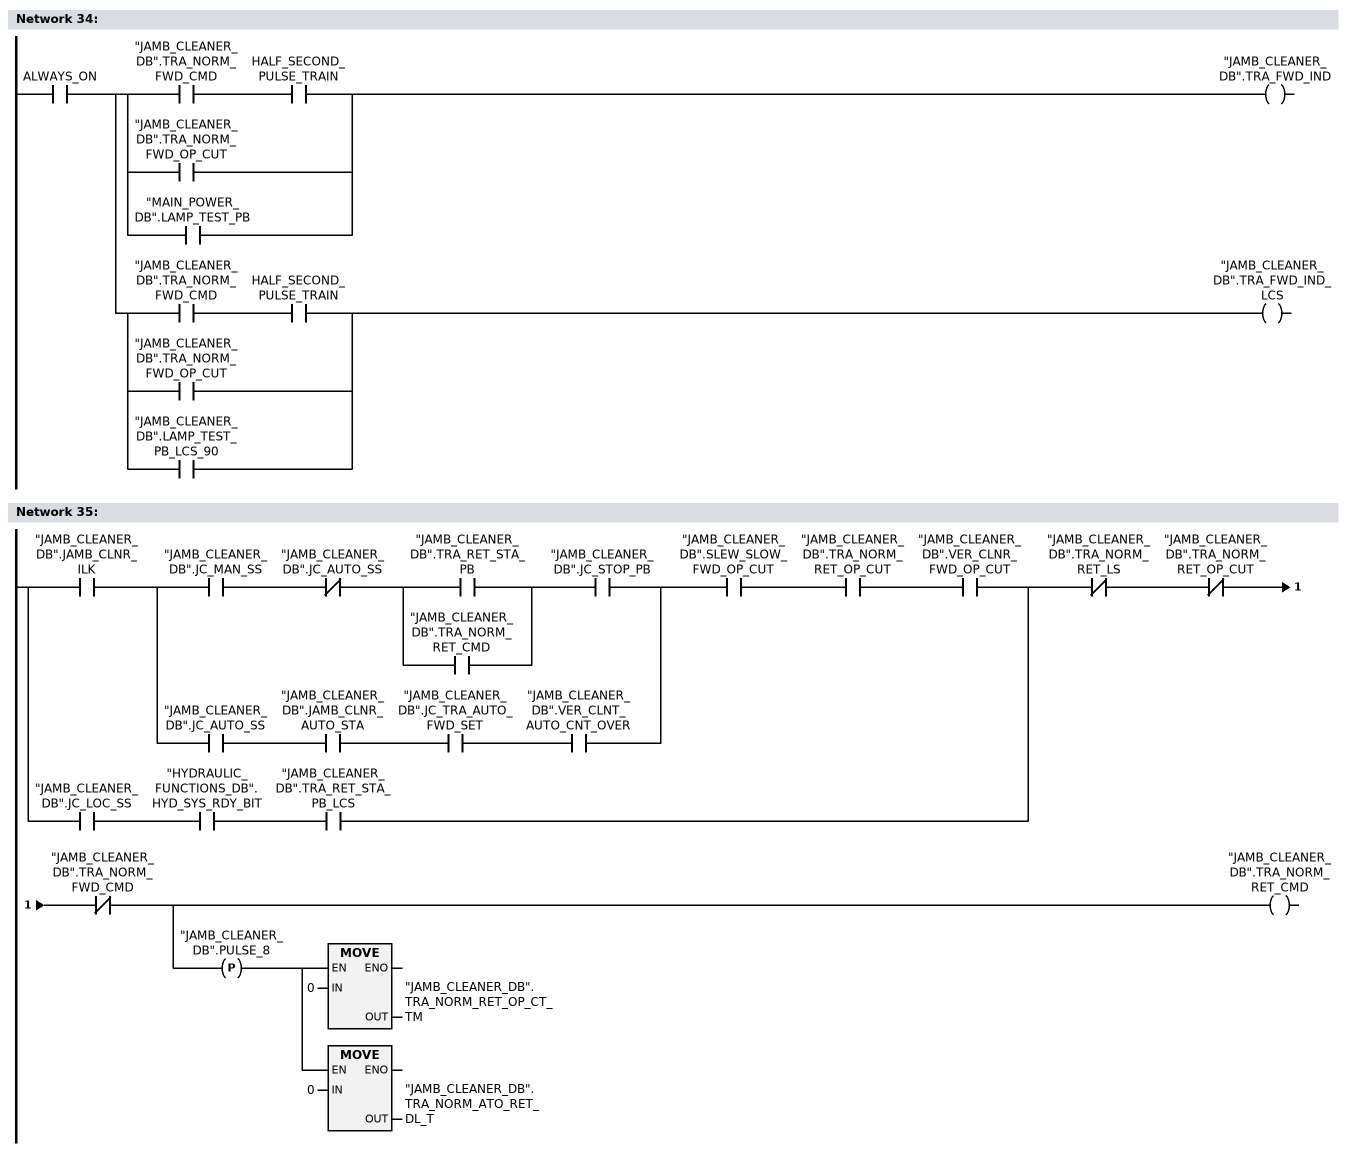
NETWORK
TITLE =
      A     "ALWAYS_ON";
      =     L 0.0;
      A     L 0.0;
      A(;
      A     "JAMB_CLEANER_DB".TRA_NORM_FWD_CMD;
      A     "HALF_SECOND_PULSE_TRAIN";
      O     "JAMB_CLEANER_DB".TRA_NORM_FWD_OP_CUT;
      O     "MAIN_POWER_DB".LAMP_TEST_PB;
      );
      =     "JAMB_CLEANER_DB".TRA_FWD_IND;
      A     L 0.0;
      A(;
      A     "JAMB_CLEANER_DB".TRA_NORM_FWD_CMD;
      A     "HALF_SECOND_PULSE_TRAIN";
      O     "JAMB_CLEANER_DB".TRA_NORM_FWD_OP_CUT;
      O     "JAMB_CLEANER_DB".LAMP_TEST_PB_LCS_90;
      );
      =     "JAMB_CLEANER_DB".TRA_FWD_IND_LCS;
NETWORK
TITLE =
      A(;
      A     "JAMB_CLEANER_DB".JAMB_CLNR_ILK;
      A(;
      A     "JAMB_CLEANER_DB".JC_MAN_SS;
      AN    "JAMB_CLEANER_DB".JC_AUTO_SS;
      A(;
      O     "JAMB_CLEANER_DB".TRA_RET_STA_PB;
      O     "JAMB_CLEANER_DB".TRA_NORM_RET_CMD;
      );
      A     "JAMB_CLEANER_DB".JC_STOP_PB;
      O;
      A     "JAMB_CLEANER_DB".JC_AUTO_SS;
      A     "JAMB_CLEANER_DB".JAMB_CLNR_AUTO_STA;
      A     "JAMB_CLEANER_DB".JC_TRA_AUTO_FWD_SET;
      A     "JAMB_CLEANER_DB".VER_CLNT_AUTO_CNT_OVER;
      );
      A     "JAMB_CLEANER_DB".SLEW_SLOW_FWD_OP_CUT;
      A     "JAMB_CLEANER_DB".TRA_NORM_RET_OP_CUT;
      A     "JAMB_CLEANER_DB".VER_CLNR_FWD_OP_CUT;
      O;
      A     "JAMB_CLEANER_DB".JC_LOC_SS;
      A     "HYDRAULIC_FUNCTIONS_DB".HYD_SYS_RDY_BIT;
      A     "JAMB_CLEANER_DB".TRA_RET_STA_PB_LCS;
      );
      AN    "JAMB_CLEANER_DB".TRA_NORM_RET_LS;
      AN    "JAMB_CLEANER_DB".TRA_NORM_RET_OP_CUT;
      AN    "JAMB_CLEANER_DB".TRA_NORM_FWD_CMD;
      =     L 0.0;
      A     L 0.0;
      BLD   102;
      =     "JAMB_CLEANER_DB".TRA_NORM_RET_CMD;
      A     L 0.0;
      FP    "JAMB_CLEANER_DB".PULSE_8;
      =     L 0.1;
      A     L 0.1;
      JNB   M030;
      L     0;
      T     "JAMB_CLEANER_DB".TRA_NORM_RET_OP_CT_TM;
M030: NOP   0;
      A     L 0.1;
      JNB   M031;
      L     0;
      T     "JAMB_CLEANER_DB".TRA_NORM_ATO_RET_DL_T;
M031: NOP   0;
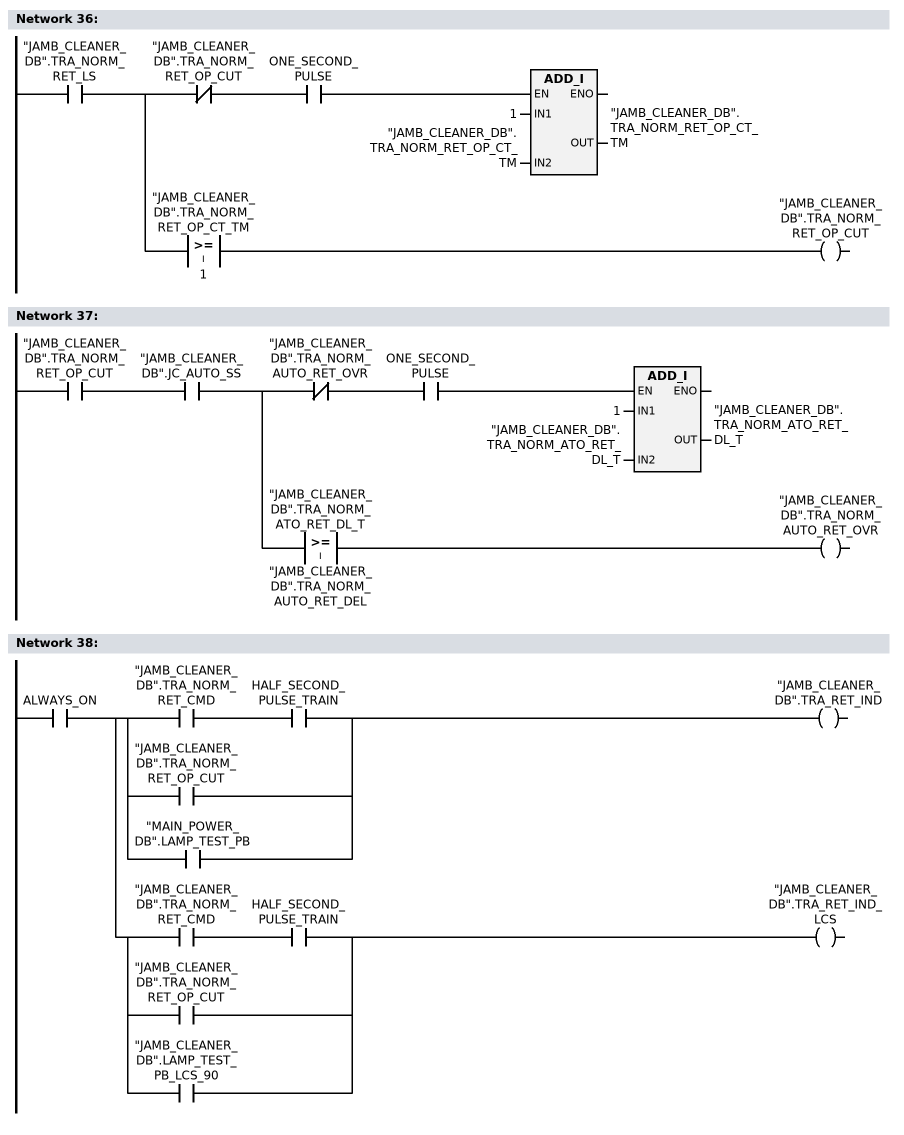
NETWORK
TITLE =
      A     "JAMB_CLEANER_DB".TRA_NORM_RET_LS;
      =     L 0.0;
      A     L 0.0;
      AN    "JAMB_CLEANER_DB".TRA_NORM_RET_OP_CUT;
      A     "ONE_SECOND_PULSE";
      JNB   M032;
      L     1;
      L     "JAMB_CLEANER_DB".TRA_NORM_RET_OP_CT_TM;
      +I;
      T     "JAMB_CLEANER_DB".TRA_NORM_RET_OP_CT_TM;
M032: NOP   0;
      A     L 0.0;
      A(;
      L     "JAMB_CLEANER_DB".TRA_NORM_RET_OP_CT_TM;
      L     1;
      >=I;
      );
      =     "JAMB_CLEANER_DB".TRA_NORM_RET_OP_CUT;
NETWORK
TITLE =
      A     "JAMB_CLEANER_DB".TRA_NORM_RET_OP_CUT;
      A     "JAMB_CLEANER_DB".JC_AUTO_SS;
      =     L 0.0;
      A     L 0.0;
      AN    "JAMB_CLEANER_DB".TRA_NORM_AUTO_RET_OVR;
      A     "ONE_SECOND_PULSE";
      JNB   M033;
      L     1;
      L     "JAMB_CLEANER_DB".TRA_NORM_ATO_RET_DL_T;
      +I;
      T     "JAMB_CLEANER_DB".TRA_NORM_ATO_RET_DL_T;
M033: NOP   0;
      A     L 0.0;
      A(;
      L     "JAMB_CLEANER_DB".TRA_NORM_ATO_RET_DL_T;
      L     "JAMB_CLEANER_DB".TRA_NORM_AUTO_RET_DEL;
      >=I;
      );
      =     "JAMB_CLEANER_DB".TRA_NORM_AUTO_RET_OVR;
NETWORK
TITLE =
      A     "ALWAYS_ON";
      =     L 0.0;
      A     L 0.0;
      A(;
      A     "JAMB_CLEANER_DB".TRA_NORM_RET_CMD;
      A     "HALF_SECOND_PULSE_TRAIN";
      O     "JAMB_CLEANER_DB".TRA_NORM_RET_OP_CUT;
      O     "MAIN_POWER_DB".LAMP_TEST_PB;
      );
      =     "JAMB_CLEANER_DB".TRA_RET_IND;
      A     L 0.0;
      A(;
      A     "JAMB_CLEANER_DB".TRA_NORM_RET_CMD;
      A     "HALF_SECOND_PULSE_TRAIN";
      O     "JAMB_CLEANER_DB".TRA_NORM_RET_OP_CUT;
      O     "JAMB_CLEANER_DB".LAMP_TEST_PB_LCS_90;
      );
      =     "JAMB_CLEANER_DB".TRA_RET_IND_LCS;
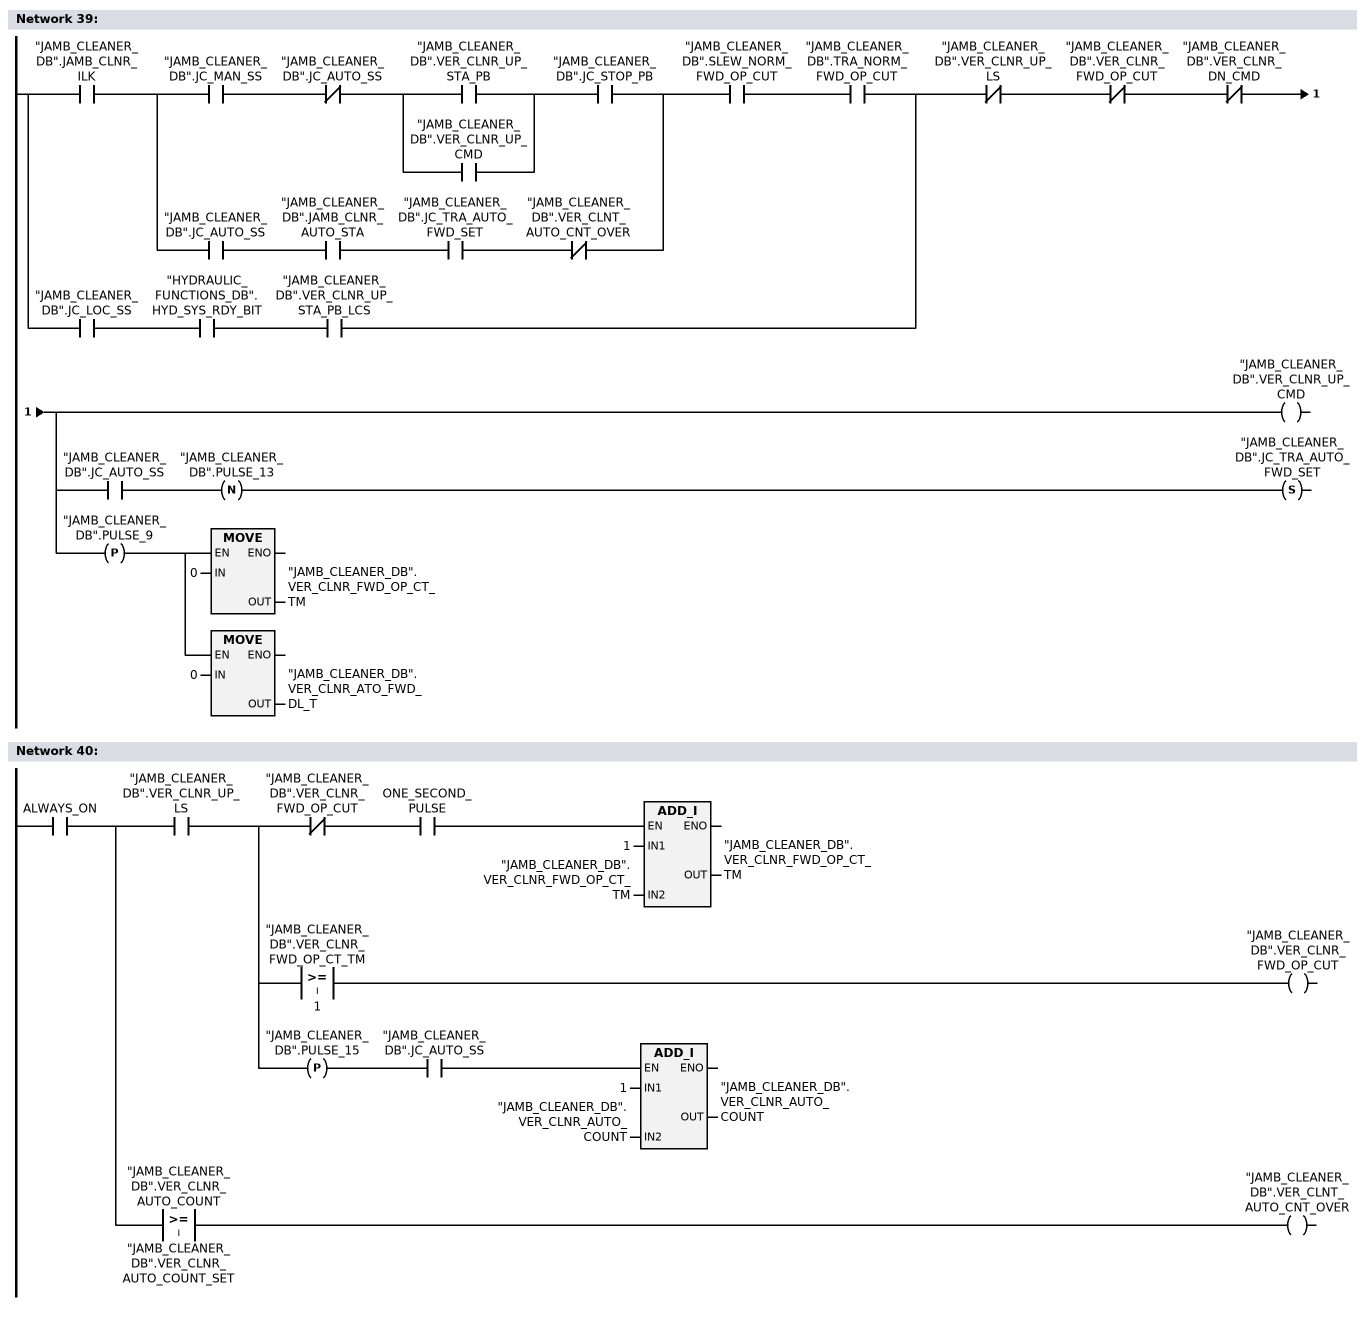
NETWORK
TITLE =
      A(;
      A     "JAMB_CLEANER_DB".JAMB_CLNR_ILK;
      A(;
      A     "JAMB_CLEANER_DB".JC_MAN_SS;
      AN    "JAMB_CLEANER_DB".JC_AUTO_SS;
      A(;
      O     "JAMB_CLEANER_DB".VER_CLNR_UP_STA_PB;
      O     "JAMB_CLEANER_DB".VER_CLNR_UP_CMD;
      );
      A     "JAMB_CLEANER_DB".JC_STOP_PB;
      O;
      A     "JAMB_CLEANER_DB".JC_AUTO_SS;
      A     "JAMB_CLEANER_DB".JAMB_CLNR_AUTO_STA;
      A     "JAMB_CLEANER_DB".JC_TRA_AUTO_FWD_SET;
      AN    "JAMB_CLEANER_DB".VER_CLNT_AUTO_CNT_OVER;
      );
      A     "JAMB_CLEANER_DB".SLEW_NORM_FWD_OP_CUT;
      A     "JAMB_CLEANER_DB".TRA_NORM_FWD_OP_CUT;
      O;
      A     "JAMB_CLEANER_DB".JC_LOC_SS;
      A     "HYDRAULIC_FUNCTIONS_DB".HYD_SYS_RDY_BIT;
      A     "JAMB_CLEANER_DB".VER_CLNR_UP_STA_PB_LCS;
      );
      AN    "JAMB_CLEANER_DB".VER_CLNR_UP_LS;
      AN    "JAMB_CLEANER_DB".VER_CLNR_FWD_OP_CUT;
      AN    "JAMB_CLEANER_DB".VER_CLNR_DN_CMD;
      =     L 0.0;
      A     L 0.0;
      BLD   102;
      =     "JAMB_CLEANER_DB".VER_CLNR_UP_CMD;
      A     L 0.0;
      A     "JAMB_CLEANER_DB".JC_AUTO_SS;
      FN    "JAMB_CLEANER_DB".PULSE_13;
      S     "JAMB_CLEANER_DB".JC_TRA_AUTO_FWD_SET;
      A     L 0.0;
      FP    "JAMB_CLEANER_DB".PULSE_9;
      =     L 0.1;
      A     L 0.1;
      JNB   M034;
      L     0;
      T     "JAMB_CLEANER_DB".VER_CLNR_FWD_OP_CT_TM;
M034: NOP   0;
      A     L 0.1;
      JNB   M035;
      L     0;
      T     "JAMB_CLEANER_DB".VER_CLNR_ATO_FWD_DL_T;
M035: NOP   0;
NETWORK
TITLE =
      A     "ALWAYS_ON";
      =     L 0.0;
      A     L 0.0;
      A     "JAMB_CLEANER_DB".VER_CLNR_UP_LS;
      =     L 0.1;
      A     L 0.1;
      AN    "JAMB_CLEANER_DB".VER_CLNR_FWD_OP_CUT;
      A     "ONE_SECOND_PULSE";
      JNB   M036;
      L     1;
      L     "JAMB_CLEANER_DB".VER_CLNR_FWD_OP_CT_TM;
      +I;
      T     "JAMB_CLEANER_DB".VER_CLNR_FWD_OP_CT_TM;
M036: NOP   0;
      A     L 0.1;
      A(;
      L     "JAMB_CLEANER_DB".VER_CLNR_FWD_OP_CT_TM;
      L     1;
      >=I;
      );
      =     "JAMB_CLEANER_DB".VER_CLNR_FWD_OP_CUT;
      A     L 0.1;
      FP    "JAMB_CLEANER_DB".PULSE_15;
      A     "JAMB_CLEANER_DB".JC_AUTO_SS;
      JNB   M037;
      L     1;
      L     "JAMB_CLEANER_DB".VER_CLNR_AUTO_COUNT;
      +I;
      T     "JAMB_CLEANER_DB".VER_CLNR_AUTO_COUNT;
M037: NOP   0;
      A     L 0.0;
      A(;
      L     "JAMB_CLEANER_DB".VER_CLNR_AUTO_COUNT;
      L     "JAMB_CLEANER_DB".VER_CLNR_AUTO_COUNT_SET;
      >=I;
      );
      =     "JAMB_CLEANER_DB".VER_CLNT_AUTO_CNT_OVER;
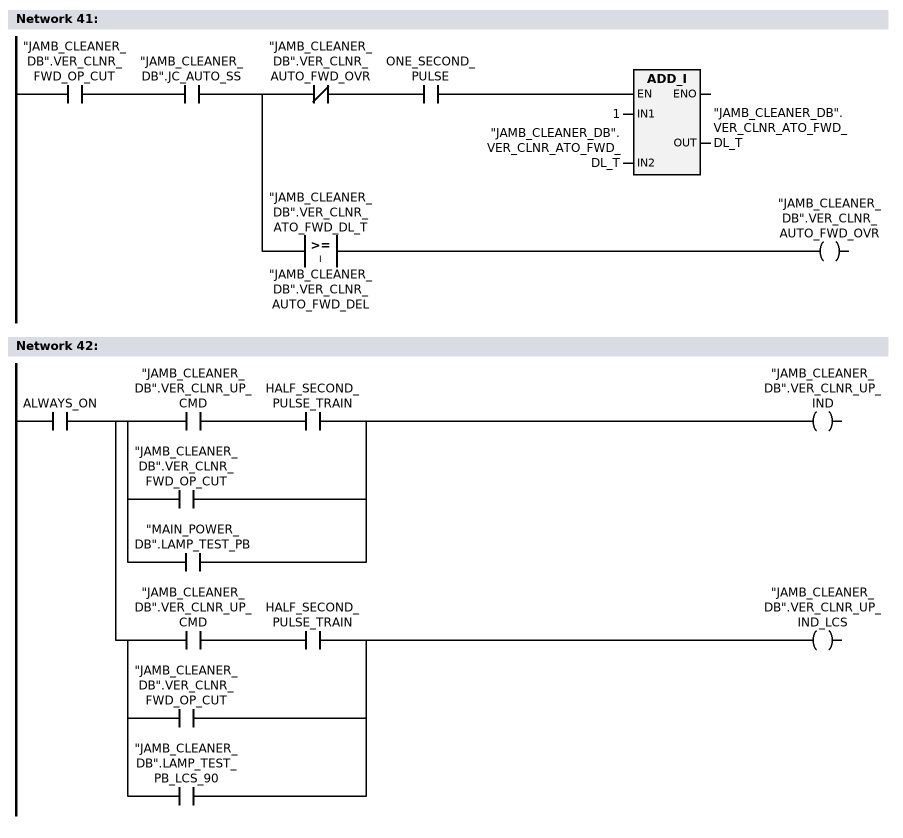
NETWORK
TITLE =
      A     "JAMB_CLEANER_DB".VER_CLNR_FWD_OP_CUT;
      A     "JAMB_CLEANER_DB".JC_AUTO_SS;
      =     L 0.0;
      A     L 0.0;
      AN    "JAMB_CLEANER_DB".VER_CLNR_AUTO_FWD_OVR;
      A     "ONE_SECOND_PULSE";
      JNB   M038;
      L     1;
      L     "JAMB_CLEANER_DB".VER_CLNR_ATO_FWD_DL_T;
      +I;
      T     "JAMB_CLEANER_DB".VER_CLNR_ATO_FWD_DL_T;
M038: NOP   0;
      A     L 0.0;
      A(;
      L     "JAMB_CLEANER_DB".VER_CLNR_ATO_FWD_DL_T;
      L     "JAMB_CLEANER_DB".VER_CLNR_AUTO_FWD_DEL;
      >=I;
      );
      =     "JAMB_CLEANER_DB".VER_CLNR_AUTO_FWD_OVR;
NETWORK
TITLE =
      A     "ALWAYS_ON";
      =     L 0.0;
      A     L 0.0;
      A(;
      A     "JAMB_CLEANER_DB".VER_CLNR_UP_CMD;
      A     "HALF_SECOND_PULSE_TRAIN";
      O     "JAMB_CLEANER_DB".VER_CLNR_FWD_OP_CUT;
      O     "MAIN_POWER_DB".LAMP_TEST_PB;
      );
      =     "JAMB_CLEANER_DB".VER_CLNR_UP_IND;
      A     L 0.0;
      A(;
      A     "JAMB_CLEANER_DB".VER_CLNR_UP_CMD;
      A     "HALF_SECOND_PULSE_TRAIN";
      O     "JAMB_CLEANER_DB".VER_CLNR_FWD_OP_CUT;
      O     "JAMB_CLEANER_DB".LAMP_TEST_PB_LCS_90;
      );
      =     "JAMB_CLEANER_DB".VER_CLNR_UP_IND_LCS;
